LIN {X 0,Y 256.536,Z 513.805,A -85,B 0,C 180,E1 -18432.463,E2 -18432.463} C_VEL
LIN {X 0,Y 255.178,Z 520.285,A -85,B 0,C 180,E1 -18435.65,E2 -18435.65} C_VEL
LIN {X 0,Y 254.431,Z 525.317,A -85,B 0,C 180,E1 -18438.853,E2 -18438.853} C_VEL
LIN {X 0,Y 254.375,Z 529.039,A -85,B 0,C 180,E1 -18442.062,E2 -18442.062} C_VEL
LIN {X 0,Y 254.585,Z 531.508,A -85,B 0,C 180,E1 -18445.252,E2 -18445.252} C_VEL
LIN {X 0,Y 254.898,Z 532.764,A -85,B 0,C 180,E1 -18448.422,E2 -18448.422} C_VEL
LIN {X 0,Y 254.986,Z 532.93,A -85,B 0,C 180,E1 -18450.002,E2 -18450.002} C_VEL
LIN {X 0,Y 254.897,Z 532.761,A -85,B 0,C 180,E1 -18451.582,E2 -18451.582} C_VEL
LIN {X 0,Y 254.605,Z 531.496,A -85,B 0,C 180,E1 -18454.752,E2 -18454.752} C_VEL
LIN {X 0,Y 254.565,Z 530.416,A -85,B 0,C 180,E1 -18456.342,E2 -18456.342} C_VEL
LIN {X 0,Y 254.406,Z 527.304,A -85,B 0,C 180,E1 -18459.543,E2 -18459.543} C_VEL
LIN {X 0,Y 254.778,Z 522.916,A -85,B 0,C 180,E1 -18462.751,E2 -18462.751} C_VEL
LIN {X 0,Y 255.788,Z 517.161,A -85,B 0,C 180,E1 -18465.95,E2 -18465.95} C_VEL
LIN {X 0,Y 257.512,Z 509.888,A -85,B 0,C 180,E1 -18469.119,E2 -18469.119} C_VEL
LIN {X 0,Y 259.708,Z 502.128,A -85,B 0,C 180,E1 -18471.847,E2 -18471.847} C_VEL
LIN {X 0,Y 262.386,Z 492.608,A -85,B 0,C 180,E1 -18474.585,E2 -18474.585} C_VEL
LIN {X 0,Y 264.113,Z 486.805,A -85,B 0,C 180,E1 -18476.046,E2 -18476.046} C_VEL
LIN {X 0,Y 268.171,Z 478.576,A -85,B 0,C 180,E1 -18478.575,E2 -18478.575} C_VEL
LIN {X 0,Y 272.785,Z 469.047,A -85,B 0,C 180,E1 -18481.018,E2 -18481.018} C_VEL
LIN {X 0,Y 278.417,Z 457.827,A -85,B 0,C 180,E1 -18483.302,E2 -18483.302} C_VEL
LIN {X 0,Y 283.318,Z 447.662,A -85,B 0,C 180,E1 -18485.029,E2 -18485.029} C_VEL
LIN {X 0,Y 289.052,Z 435.031,A -85,B 0,C 180,E1 -18486.781,E2 -18486.781} C_VEL
LIN {X 0,Y 294.359,Z 422.603,A -85,B 0,C 180,E1 -18488.156,E2 -18488.156} C_VEL
LIN {X 0,Y 300.783,Z 405.935,A -85,B 0,C 180,E1 -18489.592,E2 -18489.592} C_VEL
LIN {X 0,Y 305.874,Z 390.525,A -85,B 0,C 180,E1 -18490.616,E2 -18490.616} C_VEL
LIN {X 0,Y 310.657,Z 373.123,A -85,B 0,C 180,E1 -18491.487,E2 -18491.487} C_VEL
LIN {X 0,Y 327.276,Z 296.354,A -85,B 0,C 180,E1 -18494.561,E2 -18494.561} C_VEL
LIN {X 0,Y 328.249,Z 291.917,A -85,B 0,C 180,E1 -18494.78,E2 -18494.78} C_VEL
LIN {X 0,Y 329.621,Z 284.935,A -85,B 0,C 180,E1 -18495.368,E2 -18495.368} C_VEL
LIN {X 0,Y 329.028,Z 283.211,A -85,B 0,C 180,E1 -18497.15,E2 -18497.15} C_VEL
LIN {X 0,Y 328.897,Z 282.812,A -85,B 0,C 180,E1 -18498.516,E2 -18498.516} C_VEL
LIN {X 0,Y 328.979,Z 283.074,A -85,B 0,C 180,E1 -18499.587,E2 -18499.587} C_VEL
LIN {X 0,Y 329.408,Z 285.035,A -85,B 0,C 180,E1 -18501.432,E2 -18501.432} C_VEL
LIN {X 0,Y 316.44,Z 338.458,A -85,B 0,C 180,E1 -18503.875,E2 -18503.875} C_VEL
LIN {X 0,Y 312.736,Z 355.057,A -85,B 0,C 180,E1 -18504.791,E2 -18504.791} C_VEL
LIN {X 0,Y 309.152,Z 368.459,A -85,B 0,C 180,E1 -18505.761,E2 -18505.761} C_VEL
LIN {X 0,Y 305.253,Z 380.868,A -85,B 0,C 180,E1 -18506.878,E2 -18506.878} C_VEL
LIN {X 0,Y 300.146,Z 394.54,A -85,B 0,C 180,E1 -18508.405,E2 -18508.405} C_VEL
LIN {X 0,Y 295.293,Z 405.891,A -85,B 0,C 180,E1 -18510.013,E2 -18510.013} C_VEL
LIN {X 0,Y 290.344,Z 416.322,A -85,B 0,C 180,E1 -18511.835,E2 -18511.835} C_VEL
LIN {X 0,Y 284.968,Z 426.311,A -85,B 0,C 180,E1 -18514.039,E2 -18514.039} C_VEL
LIN {X 0,Y 280.137,Z 434.422,A -85,B 0,C 180,E1 -18516.334,E2 -18516.334} C_VEL
LIN {X 0,Y 276.27,Z 440.16,A -85,B 0,C 180,E1 -18518.355,E2 -18518.355} C_VEL
LIN {X 0,Y 272.687,Z 444.824,A -85,B 0,C 180,E1 -18520.425,E2 -18520.425} C_VEL
LIN {X 0,Y 269.52,Z 448.489,A -85,B 0,C 180,E1 -18522.55,E2 -18522.55} C_VEL
LIN {X 0,Y 266.631,Z 451.245,A -85,B 0,C 180,E1 -18524.717,E2 -18524.717} C_VEL
LIN {X 0,Y 264.88,Z 452.58,A -85,B 0,C 180,E1 -18526.185,E2 -18526.185} C_VEL
LIN {X 0,Y 261.942,Z 454.063,A -85,B 0,C 180,E1 -18529.175,E2 -18529.175} C_VEL
LIN {X 0,Y 260.72,Z 454.217,A -85,B 0,C 180,E1 -18530.692,E2 -18530.692} C_VEL
LIN {X 0,Y 259.691,Z 453.95,A -85,B 0,C 180,E1 -18532.223,E2 -18532.223} C_VEL
LIN {X 0,Y 258.915,Z 453.273,A -85,B 0,C 180,E1 -18533.767,E2 -18533.767} C_VEL
LIN {X 0,Y 258.057,Z 452.243,A -85,B 0,C 180,E1 -18535.314,E2 -18535.314} C_VEL
LIN {X 0,Y 257.5,Z 450.798,A -85,B 0,C 180,E1 -18536.871,E2 -18536.871} C_VEL
LIN {X 0,Y 256.669,Z 447.86,A -85,B 0,C 180,E1 -18539.216,E2 -18539.216} C_VEL
LIN {X 0,Y 256.295,Z 443.931,A -85,B 0,C 180,E1 -18541.572,E2 -18541.572} C_VEL
LIN {X 0,Y 256.126,Z 438.953,A -85,B 0,C 180,E1 -18543.934,E2 -18543.934} C_VEL
LIN {X 0,Y 256.246,Z 431.674,A -85,B 0,C 180,E1 -18546.694,E2 -18546.694} C_VEL
LIN {X 0,Y 256.653,Z 423.961,A -85,B 0,C 180,E1 -18549.059,E2 -18549.059} C_VEL
LIN {X 0,Y 257.214,Z 414.588,A -85,B 0,C 180,E1 -18551.426,E2 -18551.426} C_VEL
LIN {X 0,Y 258.041,Z 403.213,A -85,B 0,C 180,E1 -18553.787,E2 -18553.787} C_VEL
LIN {X 0,Y 258.858,Z 391.632,A -85,B 0,C 180,E1 -18555.754,E2 -18555.754} C_VEL
LIN {X 0,Y 259.874,Z 379.093,A -85,B 0,C 180,E1 -18557.51,E2 -18557.51} C_VEL
LIN {X 0,Y 260.674,Z 367.212,A -85,B 0,C 180,E1 -18558.877,E2 -18558.877} C_VEL
LIN {X 0,Y 261.421,Z 353.444,A -85,B 0,C 180,E1 -18560.145,E2 -18560.145} C_VEL
LIN {X 0,Y 262.078,Z 338.203,A -85,B 0,C 180,E1 -18561.225,E2 -18561.225} C_VEL
LIN {X 0,Y 262.902,Z 318.351,A -85,B 0,C 180,E1 -18562.185,E2 -18562.185} C_VEL
LIN {X 0,Y 266.851,Z 236.98,A -85,B 0,C 180,E1 -18565.669,E2 -18565.669} C_VEL
LIN {X 0,Y 263.629,Z 209.974,A -85,B 0,C 180,E1 -18567.087,E2 -18567.087} C_VEL
LIN {X 0,Y 263.411,Z 206.92,A -85,B 0,C 180,E1 -18567.274,E2 -18567.274} C_VEL
LIN {X 0,Y 263.717,Z 203.783,A -85,B 0,C 180,E1 -18568.09,E2 -18568.09} C_VEL
LIN {X 0,Y 261.466,Z 193.257,A -85,B 0,C 180,E1 -18571.159,E2 -18571.159} C_VEL
LIN {X 0,Y 258.802,Z 181.374,A -85,B 0,C 180,E1 -18574.77,E2 -18574.77} C_VEL
LIN {X 0,Y 256.106,Z 170.203,A -85,B 0,C 180,E1 -18578.385,E2 -18578.385} C_VEL
LIN {X 0,Y 256.11,Z 170.286,A -85,B 0,C 180,E1 -18579.018,E2 -18579.018} C_VEL
LIN {X 0,Y 256.597,Z 172.135,A -85,B 0,C 180,E1 -18579.554,E2 -18579.554} C_VEL
LIN {X 0,Y 260.268,Z 178.847,A -85,B 0,C 180,E1 -18581.938,E2 -18581.938} C_VEL
LIN {X 0,Y 261.702,Z 181.55,A -85,B 0,C 180,E1 -18582.76,E2 -18582.76} C_VEL
LIN {X 0,Y 270.517,Z 194.274,A -85,B 0,C 180,E1 -18585.248,E2 -18585.248} C_VEL
LIN {X 0,Y 279.32,Z 208.41,A -85,B 0,C 180,E1 -18587.531,E2 -18587.531} C_VEL
LIN {X 0,Y 286.827,Z 222.154,A -85,B 0,C 180,E1 -18589.362,E2 -18589.362} C_VEL
LIN {X 0,Y 292.137,Z 233.078,A -85,B 0,C 180,E1 -18590.609,E2 -18590.609} C_VEL
LIN {X 0,Y 289.881,Z 285.461,A -85,B 0,C 180,E1 -18591.886,E2 -18591.886} C_VEL
LIN {X 0,Y 287.05,Z 347.338,A -85,B 0,C 180,E1 -18593.413,E2 -18593.413} C_VEL
LIN {X 0,Y 285.801,Z 362.815,A -85,B 0,C 180,E1 -18594.05,E2 -18594.05} C_VEL
LIN {X 0,Y 284.285,Z 376.98,A -85,B 0,C 180,E1 -18594.916,E2 -18594.916} C_VEL
LIN {X 0,Y 282.448,Z 389.981,A -85,B 0,C 180,E1 -18595.952,E2 -18595.952} C_VEL
LIN {X 0,Y 279.884,Z 403.781,A -85,B 0,C 180,E1 -18597.323,E2 -18597.323} C_VEL
LIN {X 0,Y 277.145,Z 416.382,A -85,B 0,C 180,E1 -18598.888,E2 -18598.888} C_VEL
LIN {X 0,Y 274.351,Z 427.21,A -85,B 0,C 180,E1 -18600.495,E2 -18600.495} C_VEL
LIN {X 0,Y 271.688,Z 436.967,A -85,B 0,C 180,E1 -18602.248,E2 -18602.248} C_VEL
LIN {X 0,Y 268.811,Z 447.132,A -85,B 0,C 180,E1 -18604.442,E2 -18604.442} C_VEL
LIN {X 0,Y 265.582,Z 457.069,A -85,B 0,C 180,E1 -18607.023,E2 -18607.023} C_VEL
LIN {X 0,Y 262.901,Z 465.292,A -85,B 0,C 180,E1 -18609.662,E2 -18609.662} C_VEL
LIN {X 0,Y 260.94,Z 471.23,A -85,B 0,C 180,E1 -18611.955,E2 -18611.955} C_VEL
LIN {X 0,Y 258.75,Z 477.709,A -85,B 0,C 180,E1 -18615.045,E2 -18615.045} C_VEL
LIN {X 0,Y 257.175,Z 482.759,A -85,B 0,C 180,E1 -18618.171,E2 -18618.171} C_VEL
LIN {X 0,Y 256.121,Z 486.236,A -85,B 0,C 180,E1 -18621.059,E2 -18621.059} C_VEL
LIN {X 0,Y 255.418,Z 488.505,A -85,B 0,C 180,E1 -18623.679,E2 -18623.679} C_VEL
LIN {X 0,Y 255.12,Z 490.193,A -85,B 0,C 180,E1 -18626.84,E2 -18626.84} C_VEL
LIN {X 0,Y 254.856,Z 490.791,A -85,B 0,C 180,E1 -18629.998,E2 -18629.998} C_VEL
LIN {X 0,Y 255.117,Z 490.228,A -85,B 0,C 180,E1 -18633.156,E2 -18633.156} C_VEL
LIN {X 0,Y 255.396,Z 488.589,A -85,B 0,C 180,E1 -18636.317,E2 -18636.317} C_VEL
LIN {X 0,Y 256.28,Z 485.793,A -85,B 0,C 180,E1 -18639.468,E2 -18639.468} C_VEL
LIN {X 0,Y 257.491,Z 481.794,A -85,B 0,C 180,E1 -18642.61,E2 -18642.61} C_VEL
LIN {X 0,Y 259.2,Z 476.467,A -85,B 0,C 180,E1 -18645.73,E2 -18645.73} C_VEL
LIN {X 0,Y 261.529,Z 469.654,A -85,B 0,C 180,E1 -18648.81,E2 -18648.81} C_VEL
LIN {X 0,Y 263.766,Z 462.707,A -85,B 0,C 180,E1 -18651.367,E2 -18651.367} C_VEL
LIN {X 0,Y 266.828,Z 453.521,A -85,B 0,C 180,E1 -18654.093,E2 -18654.093} C_VEL
LIN {X 0,Y 269.685,Z 444.479,A -85,B 0,C 180,E1 -18656.294,E2 -18656.294} C_VEL
LIN {X 0,Y 272.779,Z 433.405,A -85,B 0,C 180,E1 -18658.548,E2 -18658.548} C_VEL
LIN {X 0,Y 276.079,Z 420.918,A -85,B 0,C 180,E1 -18660.603,E2 -18660.603} C_VEL
LIN {X 0,Y 279.19,Z 407.788,A -85,B 0,C 180,E1 -18662.336,E2 -18662.336} C_VEL
LIN {X 0,Y 282.032,Z 393.095,A -85,B 0,C 180,E1 -18663.885,E2 -18663.885} C_VEL
LIN {X 0,Y 284.084,Z 379.46,A -85,B 0,C 180,E1 -18665.029,E2 -18665.029} C_VEL
LIN {X 0,Y 285.771,Z 364.638,A -85,B 0,C 180,E1 -18665.972,E2 -18665.972} C_VEL
LIN {X 0,Y 287.032,Z 349.395,A -85,B 0,C 180,E1 -18666.64,E2 -18666.64} C_VEL
LIN {X 0,Y 288.549,Z 317.716,A -85,B 0,C 180,E1 -18667.453,E2 -18667.453} C_VEL
LIN {X 0,Y 292.362,Z 233.432,A -85,B 0,C 180,E1 -18669.476,E2 -18669.476} C_VEL
LIN {X 0,Y 284.919,Z 218.308,A -85,B 0,C 180,E1 -18671.239,E2 -18671.239} C_VEL
LIN {X 0,Y 275.639,Z 202.212,A -85,B 0,C 180,E1 -18673.55,E2 -18673.55} C_VEL
LIN {X 0,Y 270.298,Z 193.85,A -85,B 0,C 180,E1 -18674.963,E2 -18674.963} C_VEL
LIN {X 0,Y 266.031,Z 189.676,A -85,B 0,C 180,E1 -18676.072,E2 -18676.072} C_VEL
LIN {X 0,Y 256.851,Z 183.256,A -85,B 0,C 180,E1 -18678.535,E2 -18678.535} C_VEL
LIN {X 0,Y 254.125,Z 180.724,A -85,B 0,C 180,E1 -18679.562,E2 -18679.562} C_VEL
LIN {X 0,Y 253.472,Z 179.796,A -85,B 0,C 180,E1 -18679.924,E2 -18679.924} C_VEL
LIN {X 0,Y 251.742,Z 176.765,A -85,B 0,C 180,E1 -18681.087,E2 -18681.087} C_VEL
LIN {X 0,Y 251.149,Z 175.254,A -85,B 0,C 180,E1 -18681.581,E2 -18681.581} C_VEL
LIN {X 0,Y 249.787,Z 173.342,A -85,B 0,C 180,E1 -18682.444,E2 -18682.444} C_VEL
LIN {X 0,Y 249.075,Z 171.086,A -85,B 0,C 180,E1 -18683.245,E2 -18683.245} C_VEL
LIN {X 0,Y 249.028,Z 171.092,A -85,B 0,C 180,E1 -18687.574,E2 -18687.574} C_VEL
LIN {X 0,Y 249.092,Z 171.068,A -85,B 0,C 180,E1 -18691.338,E2 -18691.338} C_VEL
LIN {X 0,Y 249.143,Z 171.053,A -85,B 0,C 180,E1 -18694.967,E2 -18694.967} C_VEL
LIN {X 0,Y 249.1,Z 171.058,A -85,B 0,C 180,E1 -18700.21,E2 -18700.21} C_VEL
LIN {X 0,Y 249.232,Z 171.066,A -85,B 0,C 180,E1 -18703.621,E2 -18703.621} C_VEL
LIN {X 0,Y 249.243,Z 171.046,A -85,B 0,C 180,E1 -18708.616,E2 -18708.616} C_VEL
LIN {X 0,Y 249.474,Z 171.016,A -85,B 0,C 180,E1 -18711.902,E2 -18711.902} C_VEL
LIN {X 0,Y 249.428,Z 171.042,A -85,B 0,C 180,E1 -18716.769,E2 -18716.769} C_VEL
LIN {X 0,Y 249.726,Z 170.971,A -85,B 0,C 180,E1 -18720,E2 -18720} C_VEL
LIN {X 0,Y 249.428,Z 171.039,A -85,B 0,C 180,E1 -18723.23,E2 -18723.23} C_VEL
LIN {X 0,Y 249.471,Z 171.009,A -85,B 0,C 180,E1 -18728.097,E2 -18728.097} C_VEL
LIN {X 0,Y 249.242,Z 171.043,A -85,B 0,C 180,E1 -18731.384,E2 -18731.384} C_VEL
LIN {X 0,Y 249.232,Z 171.059,A -85,B 0,C 180,E1 -18736.379,E2 -18736.379} C_VEL
LIN {X 0,Y 249.077,Z 171.081,A -85,B 0,C 180,E1 -18741.519,E2 -18741.519} C_VEL
LIN {X 0,Y 249.121,Z 171.059,A -85,B 0,C 180,E1 -18745.483,E2 -18745.483} C_VEL
LIN {X 0,Y 249.064,Z 171.067,A -85,B 0,C 180,E1 -18748.99,E2 -18748.99} C_VEL
LIN {X 0,Y 249.027,Z 171.089,A -85,B 0,C 180,E1 -18752.426,E2 -18752.426} C_VEL
LIN {X 0,Y 249.075,Z 171.201,A -85,B 0,C 180,E1 -18755.337,E2 -18755.337} C_VEL
LIN {X 0,Y 250.086,Z 173.976,A -85,B 0,C 180,E1 -18755.994,E2 -18755.994} C_VEL
LIN {X 0,Y 252.285,Z 176.508,A -85,B 0,C 180,E1 -18756.961,E2 -18756.961} C_VEL
LIN {X 0,Y 254.239,Z 179.879,A -85,B 0,C 180,E1 -18757.912,E2 -18757.912} C_VEL
LIN {X 0,Y 255.171,Z 180.942,A -85,B 0,C 180,E1 -18758.294,E2 -18758.294} C_VEL
LIN {X 0,Y 257.569,Z 184.851,A -85,B 0,C 180,E1 -18759.375,E2 -18759.375} C_VEL
LIN {X 0,Y 262.205,Z 192.372,A -85,B 0,C 180,E1 -18761.319,E2 -18761.319} C_VEL
LIN {X 0,Y 268.243,Z 209.605,A -85,B 0,C 180,E1 -18764.298,E2 -18764.298} C_VEL
LIN {X 0,Y 276.939,Z 230.172,A -85,B 0,C 180,E1 -18766.8,E2 -18766.8} C_VEL
LIN {X 0,Y 280.418,Z 238.915,A -85,B 0,C 180,E1 -18767.748,E2 -18767.748} C_VEL
LIN {X 0,Y 283.617,Z 279.318,A -85,B 0,C 180,E1 -18769.64,E2 -18769.64} C_VEL
LIN {X 0,Y 284.027,Z 287.147,A -85,B 0,C 180,E1 -18769.961,E2 -18769.961} C_VEL
LIN {X 0,Y 279.389,Z 384.707,A -85,B 0,C 180,E1 -18772.356,E2 -18772.356} C_VEL
LIN {X 0,Y 277.918,Z 399.648,A -85,B 0,C 180,E1 -18772.92,E2 -18772.92} C_VEL
LIN {X 0,Y 275.926,Z 413.694,A -85,B 0,C 180,E1 -18773.69,E2 -18773.69} C_VEL
LIN {X 0,Y 273.424,Z 427.201,A -85,B 0,C 180,E1 -18774.669,E2 -18774.669} C_VEL
LIN {X 0,Y 270.251,Z 441.425,A -85,B 0,C 180,E1 -18776.008,E2 -18776.008} C_VEL
LIN {X 0,Y 266.93,Z 454.852,A -85,B 0,C 180,E1 -18777.634,E2 -18777.634} C_VEL
LIN {X 0,Y 263.299,Z 467.497,A -85,B 0,C 180,E1 -18779.528,E2 -18779.528} C_VEL
LIN {X 0,Y 260.358,Z 477.557,A -85,B 0,C 180,E1 -18781.374,E2 -18781.374} C_VEL
LIN {X 0,Y 257.208,Z 487.833,A -85,B 0,C 180,E1 -18783.642,E2 -18783.642} C_VEL
LIN {X 0,Y 254.163,Z 497.892,A -85,B 0,C 180,E1 -18786.365,E2 -18786.365} C_VEL
LIN {X 0,Y 251.623,Z 506.261,A -85,B 0,C 180,E1 -18789.14,E2 -18789.14} C_VEL
LIN {X 0,Y 249.667,Z 513.212,A -85,B 0,C 180,E1 -18791.965,E2 -18791.965} C_VEL
LIN {X 0,Y 248.228,Z 519.693,A -85,B 0,C 180,E1 -18795.24,E2 -18795.24} C_VEL
LIN {X 0,Y 247.381,Z 524.724,A -85,B 0,C 180,E1 -18798.532,E2 -18798.532} C_VEL
LIN {X 0,Y 247.292,Z 528.448,A -85,B 0,C 180,E1 -18801.833,E2 -18801.833} C_VEL
LIN {X 0,Y 247.514,Z 530.922,A -85,B 0,C 180,E1 -18805.116,E2 -18805.116} C_VEL
LIN {X 0,Y 247.811,Z 532.178,A -85,B 0,C 180,E1 -18808.377,E2 -18808.377} C_VEL
LIN {X 0,Y 247.925,Z 532.347,A -85,B 0,C 180,E1 -18810.002,E2 -18810.002} C_VEL
LIN {X 0,Y 247.81,Z 532.175,A -85,B 0,C 180,E1 -18811.627,E2 -18811.627} C_VEL
LIN {X 0,Y 247.537,Z 530.909,A -85,B 0,C 180,E1 -18814.888,E2 -18814.888} C_VEL
LIN {X 0,Y 247.462,Z 529.824,A -85,B 0,C 180,E1 -18816.525,E2 -18816.525} C_VEL
LIN {X 0,Y 247.321,Z 526.709,A -85,B 0,C 180,E1 -18819.819,E2 -18819.819} C_VEL
LIN {X 0,Y 247.763,Z 522.321,A -85,B 0,C 180,E1 -18823.118,E2 -18823.118} C_VEL
LIN {X 0,Y 248.883,Z 516.567,A -85,B 0,C 180,E1 -18826.404,E2 -18826.404} C_VEL
LIN {X 0,Y 250.729,Z 509.294,A -85,B 0,C 180,E1 -18829.657,E2 -18829.657} C_VEL
LIN {X 0,Y 253.013,Z 501.532,A -85,B 0,C 180,E1 -18832.456,E2 -18832.456} C_VEL
LIN {X 0,Y 255.792,Z 492.22,A -85,B 0,C 180,E1 -18835.207,E2 -18835.207} C_VEL
LIN {X 0,Y 256.925,Z 488.661,A -85,B 0,C 180,E1 -18836.175,E2 -18836.175} C_VEL
LIN {X 0,Y 261.341,Z 480.431,A -85,B 0,C 180,E1 -18838.953,E2 -18838.953} C_VEL
LIN {X 0,Y 266.061,Z 471.495,A -85,B 0,C 180,E1 -18841.448,E2 -18841.448} C_VEL
LIN {X 0,Y 271.832,Z 461.11,A -85,B 0,C 180,E1 -18843.772,E2 -18843.772} C_VEL
LIN {X 0,Y 277.172,Z 450.863,A -85,B 0,C 180,E1 -18845.677,E2 -18845.677} C_VEL
LIN {X 0,Y 283.089,Z 439.038,A -85,B 0,C 180,E1 -18847.464,E2 -18847.464} C_VEL
LIN {X 0,Y 289.615,Z 425.159,A -85,B 0,C 180,E1 -18849.121,E2 -18849.121} C_VEL
LIN {X 0,Y 296.704,Z 408.403,A -85,B 0,C 180,E1 -18850.648,E2 -18850.648} C_VEL
LIN {X 0,Y 302.336,Z 393.002,A -85,B 0,C 180,E1 -18851.715,E2 -18851.715} C_VEL
LIN {X 0,Y 307.881,Z 374.881,A -85,B 0,C 180,E1 -18852.664,E2 -18852.664} C_VEL
LIN {X 0,Y 313.284,Z 351.402,A -85,B 0,C 180,E1 -18853.632,E2 -18853.632} C_VEL
LIN {X 0,Y 326.613,Z 294.43,A -85,B 0,C 180,E1 -18855.907,E2 -18855.907} C_VEL
LIN {X 0,Y 327.357,Z 290.873,A -85,B 0,C 180,E1 -18856.23,E2 -18856.23} C_VEL
LIN {X 0,Y 327.092,Z 289.871,A -85,B 0,C 180,E1 -18857.46,E2 -18857.46} C_VEL
LIN {X 0,Y 327.032,Z 289.726,A -85,B 0,C 180,E1 -18859.296,E2 -18859.296} C_VEL
LIN {X 0,Y 327.104,Z 290.812,A -85,B 0,C 180,E1 -18860.396,E2 -18860.396} C_VEL
LIN {X 0,Y 313.508,Z 344.767,A -85,B 0,C 180,E1 -18862.903,E2 -18862.903} C_VEL
LIN {X 0,Y 310.152,Z 358.542,A -85,B 0,C 180,E1 -18863.702,E2 -18863.702} C_VEL
LIN {X 0,Y 305.497,Z 374.231,A -85,B 0,C 180,E1 -18864.892,E2 -18864.892} C_VEL
LIN {X 0,Y 300.968,Z 386.739,A -85,B 0,C 180,E1 -18866.116,E2 -18866.116} C_VEL
LIN {X 0,Y 295.592,Z 399.622,A -85,B 0,C 180,E1 -18867.659,E2 -18867.659} C_VEL
LIN {X 0,Y 290.065,Z 411.145,A -85,B 0,C 180,E1 -18869.416,E2 -18869.416} C_VEL
LIN {X 0,Y 284.888,Z 420.753,A -85,B 0,C 180,E1 -18871.246,E2 -18871.246} C_VEL
LIN {X 0,Y 280.059,Z 428.908,A -85,B 0,C 180,E1 -18873.147,E2 -18873.147} C_VEL
LIN {X 0,Y 275.65,Z 435.696,A -85,B 0,C 180,E1 -18875.122,E2 -18875.122} C_VEL
LIN {X 0,Y 271.474,Z 441.357,A -85,B 0,C 180,E1 -18877.15,E2 -18877.15} C_VEL
LIN {X 0,Y 267.638,Z 446.047,A -85,B 0,C 180,E1 -18879.237,E2 -18879.237} C_VEL
LIN {X 0,Y 264.173,Z 449.709,A -85,B 0,C 180,E1 -18881.383,E2 -18881.383} C_VEL
LIN {X 0,Y 260.072,Z 453.216,A -85,B 0,C 180,E1 -18884.322,E2 -18884.322} C_VEL
LIN {X 0,Y 258.236,Z 454.39,A -85,B 0,C 180,E1 -18885.822,E2 -18885.822} C_VEL
LIN {X 0,Y 255.125,Z 455.511,A -85,B 0,C 180,E1 -18888.882,E2 -18888.882} C_VEL
LIN {X 0,Y 253.832,Z 455.496,A -85,B 0,C 180,E1 -18890.438,E2 -18890.438} C_VEL
LIN {X 0,Y 251.953,Z 454.272,A -85,B 0,C 180,E1 -18893.594,E2 -18893.594} C_VEL
LIN {X 0,Y 251.059,Z 453.11,A -85,B 0,C 180,E1 -18895.183,E2 -18895.183} C_VEL
LIN {X 0,Y 250.13,Z 450.551,A -85,B 0,C 180,E1 -18897.585,E2 -18897.585} C_VEL
LIN {X 0,Y 249.344,Z 447.068,A -85,B 0,C 180,E1 -18900,E2 -18900} C_VEL
LIN {X 0,Y 249.111,Z 442.563,A -85,B 0,C 180,E1 -18902.426,E2 -18902.426} C_VEL
LIN {X 0,Y 249.031,Z 435.932,A -85,B 0,C 180,E1 -18905.263,E2 -18905.263} C_VEL
LIN {X 0,Y 249.417,Z 427.545,A -85,B 0,C 180,E1 -18908.099,E2 -18908.099} C_VEL
LIN {X 0,Y 249.843,Z 418.719,A -85,B 0,C 180,E1 -18910.535,E2 -18910.535} C_VEL
LIN {X 0,Y 250.622,Z 408.042,A -85,B 0,C 180,E1 -18912.964,E2 -18912.964} C_VEL
LIN {X 0,Y 251.508,Z 396.079,A -85,B 0,C 180,E1 -18915.187,E2 -18915.187} C_VEL
LIN {X 0,Y 252.395,Z 384.282,A -85,B 0,C 180,E1 -18917,E2 -18917} C_VEL
LIN {X 0,Y 253.536,Z 369.719,A -85,B 0,C 180,E1 -18918.799,E2 -18918.799} C_VEL
LIN {X 0,Y 254.275,Z 355.561,A -85,B 0,C 180,E1 -18920.189,E2 -18920.189} C_VEL
LIN {X 0,Y 255.037,Z 339.802,A -85,B 0,C 180,E1 -18921.363,E2 -18921.363} C_VEL
LIN {X 0,Y 255.684,Z 323.748,A -85,B 0,C 180,E1 -18922.207,E2 -18922.207} C_VEL
LIN {X 0,Y 259.997,Z 238.073,A -85,B 0,C 180,E1 -18926.006,E2 -18926.006} C_VEL
LIN {X 0,Y 256.816,Z 210.902,A -85,B 0,C 180,E1 -18927.469,E2 -18927.469} C_VEL
LIN {X 0,Y 256.568,Z 207.28,A -85,B 0,C 180,E1 -18927.683,E2 -18927.683} C_VEL
LIN {X 0,Y 256.729,Z 204.889,A -85,B 0,C 180,E1 -18928.328,E2 -18928.328} C_VEL
LIN {X 0,Y 254.286,Z 193.66,A -85,B 0,C 180,E1 -18931.677,E2 -18931.677} C_VEL
LIN {X 0,Y 252.016,Z 183.382,A -85,B 0,C 180,E1 -18934.868,E2 -18934.868} C_VEL
LIN {X 0,Y 249.804,Z 174.098,A -85,B 0,C 180,E1 -18937.921,E2 -18937.921} C_VEL
LIN {X 0,Y 251.531,Z 176.347,A -85,B 0,C 180,E1 -18938.952,E2 -18938.952} C_VEL
LIN {X 0,Y 254.556,Z 182.21,A -85,B 0,C 180,E1 -18940.987,E2 -18940.987} C_VEL
LIN {X 0,Y 260.072,Z 189.785,A -85,B 0,C 180,E1 -18942.697,E2 -18942.697} C_VEL
LIN {X 0,Y 267.015,Z 199.952,A -85,B 0,C 180,E1 -18944.701,E2 -18944.701} C_VEL
LIN {X 0,Y 275.207,Z 213.371,A -85,B 0,C 180,E1 -18946.904,E2 -18946.904} C_VEL
LIN {X 0,Y 282.388,Z 226.708,A -85,B 0,C 180,E1 -18948.723,E2 -18948.723} C_VEL
LIN {X 0,Y 286.681,Z 235.63,A -85,B 0,C 180,E1 -18949.775,E2 -18949.775} C_VEL
LIN {X 0,Y 283.811,Z 296.33,A -85,B 0,C 180,E1 -18951.25,E2 -18951.25} C_VEL
LIN {X 0,Y 281.398,Z 347.863,A -85,B 0,C 180,E1 -18952.554,E2 -18952.554} C_VEL
LIN {X 0,Y 280.165,Z 362.884,A -85,B 0,C 180,E1 -18953.178,E2 -18953.178} C_VEL
LIN {X 0,Y 278.675,Z 376.502,A -85,B 0,C 180,E1 -18954.009,E2 -18954.009} C_VEL
LIN {X 0,Y 276.62,Z 390.551,A -85,B 0,C 180,E1 -18955.133,E2 -18955.133} C_VEL
LIN {X 0,Y 273.976,Z 404.354,A -85,B 0,C 180,E1 -18956.527,E2 -18956.527} C_VEL
LIN {X 0,Y 271.126,Z 416.958,A -85,B 0,C 180,E1 -18958.118,E2 -18958.118} C_VEL
LIN {X 0,Y 268.208,Z 427.791,A -85,B 0,C 180,E1 -18959.749,E2 -18959.749} C_VEL
LIN {X 0,Y 265.435,Z 437.55,A -85,B 0,C 180,E1 -18961.535,E2 -18961.535} C_VEL
LIN {X 0,Y 262.446,Z 447.714,A -85,B 0,C 180,E1 -18963.776,E2 -18963.776} C_VEL
LIN {X 0,Y 259.085,Z 457.652,A -85,B 0,C 180,E1 -18966.413,E2 -18966.413} C_VEL
LIN {X 0,Y 256.26,Z 465.877,A -85,B 0,C 180,E1 -18969.111,E2 -18969.111} C_VEL
LIN {X 0,Y 254.2,Z 471.816,A -85,B 0,C 180,E1 -18971.459,E2 -18971.459} C_VEL
LIN {X 0,Y 251.917,Z 478.294,A -85,B 0,C 180,E1 -18974.629,E2 -18974.629} C_VEL
LIN {X 0,Y 250.244,Z 483.345,A -85,B 0,C 180,E1 -18977.838,E2 -18977.838} C_VEL
LIN {X 0,Y 249.111,Z 486.928,A -85,B 0,C 180,E1 -18980.908,E2 -18980.908} C_VEL
LIN {X 0,Y 248.384,Z 489.09,A -85,B 0,C 180,E1 -18983.499,E2 -18983.499} C_VEL
LIN {X 0,Y 248.079,Z 490.776,A -85,B 0,C 180,E1 -18986.75,E2 -18986.75} C_VEL
LIN {X 0,Y 247.803,Z 491.374,A -85,B 0,C 180,E1 -18989.998,E2 -18989.998} C_VEL
LIN {X 0,Y 248.076,Z 490.811,A -85,B 0,C 180,E1 -18993.246,E2 -18993.246} C_VEL
LIN {X 0,Y 248.364,Z 489.173,A -85,B 0,C 180,E1 -18996.497,E2 -18996.497} C_VEL
LIN {X 0,Y 249.293,Z 486.378,A -85,B 0,C 180,E1 -18999.736,E2 -18999.736} C_VEL
LIN {X 0,Y 250.579,Z 482.378,A -85,B 0,C 180,E1 -19002.964,E2 -19002.964} C_VEL
LIN {X 0,Y 252.388,Z 477.05,A -85,B 0,C 180,E1 -19006.166,E2 -19006.166} C_VEL
LIN {X 0,Y 254.83,Z 470.236,A -85,B 0,C 180,E1 -19009.324,E2 -19009.324} C_VEL
LIN {X 0,Y 257.302,Z 462.912,A -85,B 0,C 180,E1 -19012.065,E2 -19012.065} C_VEL
LIN {X 0,Y 260.367,Z 454.101,A -85,B 0,C 180,E1 -19014.73,E2 -19014.73} C_VEL
LIN {X 0,Y 263.36,Z 445.056,A -85,B 0,C 180,E1 -19016.976,E2 -19016.976} C_VEL
LIN {X 0,Y 266.516,Z 434.189,A -85,B 0,C 180,E1 -19019.235,E2 -19019.235} C_VEL
LIN {X 0,Y 269.713,Z 422.629,A -85,B 0,C 180,E1 -19021.188,E2 -19021.188} C_VEL
LIN {X 0,Y 272.887,Z 409.752,A -85,B 0,C 180,E1 -19022.958,E2 -19022.958} C_VEL
LIN {X 0,Y 275.522,Z 397.187,A -85,B 0,C 180,E1 -19024.355,E2 -19024.355} C_VEL
LIN {X 0,Y 277.864,Z 383.592,A -85,B 0,C 180,E1 -19025.57,E2 -19025.57} C_VEL
LIN {X 0,Y 279.622,Z 369.146,A -85,B 0,C 180,E1 -19026.593,E2 -19026.593} C_VEL
LIN {X 0,Y 281.057,Z 354.334,A -85,B 0,C 180,E1 -19027.326,E2 -19027.326} C_VEL
LIN {X 0,Y 282.01,Z 337.753,A -85,B 0,C 180,E1 -19027.853,E2 -19027.853} C_VEL
LIN {X 0,Y 286.823,Z 235.74,A -85,B 0,C 180,E1 -19030.333,E2 -19030.333} C_VEL
LIN {X 0,Y 279.234,Z 220.529,A -85,B 0,C 180,E1 -19032.21,E2 -19032.21} C_VEL
LIN {X 0,Y 270.912,Z 206.138,A -85,B 0,C 180,E1 -19034.379,E2 -19034.379} C_VEL
LIN {X 0,Y 263.553,Z 194.732,A -85,B 0,C 180,E1 -19036.436,E2 -19036.436} C_VEL
LIN {X 0,Y 256.118,Z 184.27,A -85,B 0,C 180,E1 -19038.681,E2 -19038.681} C_VEL
LIN {X 0,Y 254.314,Z 181.772,A -85,B 0,C 180,E1 -19039.284,E2 -19039.284} C_VEL
LIN {X 0,Y 253.472,Z 179.796,A -85,B 0,C 180,E1 -19039.924,E2 -19039.924} C_VEL
LIN {X 0,Y 251.945,Z 178.354,A -85,B 0,C 180,E1 -19040.686,E2 -19040.686} C_VEL
LIN {X 0,Y 248.463,Z 177.34,A -85,B 0,C 180,E1 -19041.976,E2 -19041.976} C_VEL
LIN {X 0,Y 244.957,Z 176.469,A -85,B 0,C 180,E1 -19043.305,E2 -19043.305} C_VEL
LIN {X 0,Y 243.397,Z 175.229,A -85,B 0,C 180,E1 -19044.123,E2 -19044.123} C_VEL
LIN {X 0,Y 242.265,Z 173.058,A -85,B 0,C 180,E1 -19045.044,E2 -19045.044} C_VEL
LIN {X 0,Y 242.03,Z 171.944,A -85,B 0,C 180,E1 -19045.448,E2 -19045.448} C_VEL
LIN {X 0,Y 242.03,Z 171.942,A -85,B 0,C 180,E1 -19050.585,E2 -19050.585} C_VEL
LIN {X 0,Y 242.059,Z 171.94,A -85,B 0,C 180,E1 -19054.182,E2 -19054.182} C_VEL
LIN {X 0,Y 242.044,Z 171.961,A -85,B 0,C 180,E1 -19058.296,E2 -19058.296} C_VEL
LIN {X 0,Y 242.154,Z 171.942,A -85,B 0,C 180,E1 -19063.277,E2 -19063.277} C_VEL
LIN {X 0,Y 242.176,Z 171.921,A -85,B 0,C 180,E1 -19068.279,E2 -19068.279} C_VEL
LIN {X 0,Y 242.425,Z 171.897,A -85,B 0,C 180,E1 -19071.665,E2 -19071.665} C_VEL
LIN {X 0,Y 242.251,Z 171.913,A -85,B 0,C 180,E1 -19075.007,E2 -19075.007} C_VEL
LIN {X 0,Y 242.627,Z 171.871,A -85,B 0,C 180,E1 -19078.34,E2 -19078.34} C_VEL
LIN {X 0,Y 242.627,Z 171.864,A -85,B 0,C 180,E1 -19081.66,E2 -19081.66} C_VEL
LIN {X 0,Y 242.424,Z 171.879,A -85,B 0,C 180,E1 -19086.659,E2 -19086.659} C_VEL
LIN {X 0,Y 242.304,Z 171.923,A -85,B 0,C 180,E1 -19090.022,E2 -19090.022} C_VEL
LIN {X 0,Y 242.156,Z 171.931,A -85,B 0,C 180,E1 -19095.141,E2 -19095.141} C_VEL
LIN {X 0,Y 242.063,Z 171.928,A -85,B 0,C 180,E1 -19098.625,E2 -19098.625} C_VEL
LIN {X 0,Y 242.003,Z 171.962,A -85,B 0,C 180,E1 -19102.181,E2 -19102.181} C_VEL
LIN {X 0,Y 242.057,Z 171.942,A -85,B 0,C 180,E1 -19105.839,E2 -19105.839} C_VEL
LIN {X 0,Y 241.998,Z 171.945,A -85,B 0,C 180,E1 -19109.584,E2 -19109.584} C_VEL
LIN {X 0,Y 241.973,Z 172.039,A -85,B 0,C 180,E1 -19113.015,E2 -19113.015} C_VEL
LIN {X 0,Y 243.096,Z 174.98,A -85,B 0,C 180,E1 -19113.816,E2 -19113.816} C_VEL
LIN {X 0,Y 245.408,Z 177.662,A -85,B 0,C 180,E1 -19114.943,E2 -19114.943} C_VEL
LIN {X 0,Y 247.382,Z 180.974,A -85,B 0,C 180,E1 -19115.992,E2 -19115.992} C_VEL
LIN {X 0,Y 248.404,Z 182.138,A -85,B 0,C 180,E1 -19116.452,E2 -19116.452} C_VEL
LIN {X 0,Y 250.802,Z 185.973,A -85,B 0,C 180,E1 -19117.615,E2 -19117.615} C_VEL
LIN {X 0,Y 256.362,Z 194.76,A -85,B 0,C 180,E1 -19120.107,E2 -19120.107} C_VEL
LIN {X 0,Y 257.933,Z 197.915,A -85,B 0,C 180,E1 -19120.839,E2 -19120.839} C_VEL
LIN {X 0,Y 261.667,Z 208.915,A -85,B 0,C 180,E1 -19122.799,E2 -19122.799} C_VEL
LIN {X 0,Y 267.711,Z 222.786,A -85,B 0,C 180,E1 -19124.673,E2 -19124.673} C_VEL
LIN {X 0,Y 275.279,Z 241.482,A -85,B 0,C 180,E1 -19126.874,E2 -19126.874} C_VEL
LIN {X 0,Y 278.586,Z 285.723,A -85,B 0,C 180,E1 -19128.982,E2 -19128.982} C_VEL
LIN {X 0,Y 273.991,Z 381.324,A -85,B 0,C 180,E1 -19131.363,E2 -19131.363} C_VEL
LIN {X 0,Y 272.643,Z 396.433,A -85,B 0,C 180,E1 -19131.902,E2 -19131.902} C_VEL
LIN {X 0,Y 270.644,Z 410.578,A -85,B 0,C 180,E1 -19132.63,E2 -19132.63} C_VEL
LIN {X 0,Y 268.087,Z 424.672,A -85,B 0,C 180,E1 -19133.624,E2 -19133.624} C_VEL
LIN {X 0,Y 264.757,Z 439.279,A -85,B 0,C 180,E1 -19134.97,E2 -19134.97} C_VEL
LIN {X 0,Y 261.551,Z 451.91,A -85,B 0,C 180,E1 -19136.463,E2 -19136.463} C_VEL
LIN {X 0,Y 257.911,Z 464.78,A -85,B 0,C 180,E1 -19138.364,E2 -19138.364} C_VEL
LIN {X 0,Y 254.611,Z 475.065,A -85,B 0,C 180,E1 -19140.211,E2 -19140.211} C_VEL
LIN {X 0,Y 251.289,Z 485.608,A -85,B 0,C 180,E1 -19142.521,E2 -19142.521} C_VEL
LIN {X 0,Y 248.047,Z 495.609,A -85,B 0,C 180,E1 -19145.193,E2 -19145.193} C_VEL
LIN {X 0,Y 245.288,Z 504.537,A -85,B 0,C 180,E1 -19148.134,E2 -19148.134} C_VEL
LIN {X 0,Y 242.815,Z 512.619,A -85,B 0,C 180,E1 -19151.437,E2 -19151.437} C_VEL
LIN {X 0,Y 241.265,Z 519.1,A -85,B 0,C 180,E1 -19154.804,E2 -19154.804} C_VEL
LIN {X 0,Y 240.339,Z 524.131,A -85,B 0,C 180,E1 -19158.191,E2 -19158.191} C_VEL
LIN {X 0,Y 240.189,Z 527.856,A -85,B 0,C 180,E1 -19161.59,E2 -19161.59} C_VEL
LIN {X 0,Y 240.422,Z 530.334,A -85,B 0,C 180,E1 -19164.971,E2 -19164.971} C_VEL
LIN {X 0,Y 240.726,Z 531.592,A -85,B 0,C 180,E1 -19168.329,E2 -19168.329} C_VEL
LIN {X 0,Y 240.864,Z 531.763,A -85,B 0,C 180,E1 -19170.002,E2 -19170.002} C_VEL
LIN {X 0,Y 240.726,Z 531.589,A -85,B 0,C 180,E1 -19171.675,E2 -19171.675} C_VEL
LIN {X 0,Y 240.446,Z 530.321,A -85,B 0,C 180,E1 -19175.033,E2 -19175.033} C_VEL
LIN {X 0,Y 240.352,Z 529.233,A -85,B 0,C 180,E1 -19176.719,E2 -19176.719} C_VEL
LIN {X 0,Y 240.255,Z 526.116,A -85,B 0,C 180,E1 -19180.111,E2 -19180.111} C_VEL
LIN {X 0,Y 240.761,Z 521.727,A -85,B 0,C 180,E1 -19183.507,E2 -19183.507} C_VEL
LIN {X 0,Y 241.966,Z 515.971,A -85,B 0,C 180,E1 -19186.887,E2 -19186.887} C_VEL
LIN {X 0,Y 243.937,Z 508.697,A -85,B 0,C 180,E1 -19190.228,E2 -19190.228} C_VEL
LIN {X 0,Y 246.359,Z 500.937,A -85,B 0,C 180,E1 -19193.097,E2 -19193.097} C_VEL
LIN {X 0,Y 249.546,Z 490.893,A -85,B 0,C 180,E1 -19196.109,E2 -19196.109} C_VEL
LIN {X 0,Y 254.49,Z 482.168,A -85,B 0,C 180,E1 -19199.355,E2 -19199.355} C_VEL
LIN {X 0,Y 260.101,Z 472.572,A -85,B 0,C 180,E1 -19202.254,E2 -19202.254} C_VEL
LIN {X 0,Y 266.952,Z 461.181,A -85,B 0,C 180,E1 -19204.934,E2 -19204.934} C_VEL
LIN {X 0,Y 272.592,Z 451.213,A -85,B 0,C 180,E1 -19206.831,E2 -19206.831} C_VEL
LIN {X 0,Y 278.792,Z 439.861,A -85,B 0,C 180,E1 -19208.605,E2 -19208.605} C_VEL
LIN {X 0,Y 285.563,Z 426.579,A -85,B 0,C 180,E1 -19210.246,E2 -19210.246} C_VEL
LIN {X 0,Y 292.284,Z 412.067,A -85,B 0,C 180,E1 -19211.626,E2 -19211.626} C_VEL
LIN {X 0,Y 298.69,Z 396.357,A -85,B 0,C 180,E1 -19212.787,E2 -19212.787} C_VEL
LIN {X 0,Y 303.757,Z 381.793,A -85,B 0,C 180,E1 -19213.614,E2 -19213.614} C_VEL
LIN {X 0,Y 308.669,Z 364.598,A -85,B 0,C 180,E1 -19214.383,E2 -19214.383} C_VEL
LIN {X 0,Y 325.261,Z 297.037,A -85,B 0,C 180,E1 -19217.054,E2 -19217.054} C_VEL
LIN {X 0,Y 325.113,Z 296.581,A -85,B 0,C 180,E1 -19217.923,E2 -19217.923} C_VEL
LIN {X 0,Y 325.11,Z 296.665,A -85,B 0,C 180,E1 -19219.372,E2 -19219.372} C_VEL
LIN {X 0,Y 311.551,Z 348.188,A -85,B 0,C 180,E1 -19221.762,E2 -19221.762} C_VEL
LIN {X 0,Y 307.916,Z 361.828,A -85,B 0,C 180,E1 -19222.577,E2 -19222.577} C_VEL
LIN {X 0,Y 303.582,Z 375.43,A -85,B 0,C 180,E1 -19223.614,E2 -19223.614} C_VEL
LIN {X 0,Y 298.765,Z 387.827,A -85,B 0,C 180,E1 -19224.808,E2 -19224.808} C_VEL
LIN {X 0,Y 293.069,Z 400.582,A -85,B 0,C 180,E1 -19226.32,E2 -19226.32} C_VEL
LIN {X 0,Y 286.727,Z 412.918,A -85,B 0,C 180,E1 -19228.198,E2 -19228.198} C_VEL
LIN {X 0,Y 280.367,Z 423.832,A -85,B 0,C 180,E1 -19230.325,E2 -19230.325} C_VEL
LIN {X 0,Y 274.461,Z 432.735,A -85,B 0,C 180,E1 -19232.554,E2 -19232.554} C_VEL
LIN {X 0,Y 269.834,Z 439.049,A -85,B 0,C 180,E1 -19234.548,E2 -19234.548} C_VEL
LIN {X 0,Y 265.458,Z 444.379,A -85,B 0,C 180,E1 -19236.602,E2 -19236.602} C_VEL
LIN {X 0,Y 260.162,Z 449.91,A -85,B 0,C 180,E1 -19239.441,E2 -19239.441} C_VEL
LIN {X 0,Y 255.577,Z 453.8,A -85,B 0,C 180,E1 -19242.393,E2 -19242.393} C_VEL
LIN {X 0,Y 251.576,Z 456.113,A -85,B 0,C 180,E1 -19245.438,E2 -19245.438} C_VEL
LIN {X 0,Y 248.304,Z 456.923,A -85,B 0,C 180,E1 -19248.573,E2 -19248.573} C_VEL
LIN {X 0,Y 245.836,Z 456.2,A -85,B 0,C 180,E1 -19251.782,E2 -19251.782} C_VEL
LIN {X 0,Y 244.972,Z 455.218,A -85,B 0,C 180,E1 -19253.411,E2 -19253.411} C_VEL
LIN {X 0,Y 244.042,Z 453.871,A -85,B 0,C 180,E1 -19255.044,E2 -19255.044} C_VEL
LIN {X 0,Y 243.063,Z 451.116,A -85,B 0,C 180,E1 -19257.514,E2 -19257.514} C_VEL
LIN {X 0,Y 242.253,Z 447.413,A -85,B 0,C 180,E1 -19260,E2 -19260} C_VEL
LIN {X 0,Y 242.018,Z 442.667,A -85,B 0,C 180,E1 -19262.497,E2 -19262.497} C_VEL
LIN {X 0,Y 241.949,Z 435.701,A -85,B 0,C 180,E1 -19265.417,E2 -19265.417} C_VEL
LIN {X 0,Y 242.368,Z 426.997,A -85,B 0,C 180,E1 -19268.337,E2 -19268.337} C_VEL
LIN {X 0,Y 242.834,Z 417.837,A -85,B 0,C 180,E1 -19270.843,E2 -19270.843} C_VEL
LIN {X 0,Y 243.632,Z 406.701,A -85,B 0,C 180,E1 -19273.343,E2 -19273.343} C_VEL
LIN {X 0,Y 244.486,Z 395.526,A -85,B 0,C 180,E1 -19275.421,E2 -19275.421} C_VEL
LIN {X 0,Y 245.439,Z 383.378,A -85,B 0,C 180,E1 -19277.283,E2 -19277.283} C_VEL
LIN {X 0,Y 246.46,Z 370.286,A -85,B 0,C 180,E1 -19278.927,E2 -19278.927} C_VEL
LIN {X 0,Y 247.158,Z 357.689,A -85,B 0,C 180,E1 -19280.217,E2 -19280.217} C_VEL
LIN {X 0,Y 247.934,Z 342.665,A -85,B 0,C 180,E1 -19281.405,E2 -19281.405} C_VEL
LIN {X 0,Y 248.512,Z 328.59,A -85,B 0,C 180,E1 -19282.226,E2 -19282.226} C_VEL
LIN {X 0,Y 252.287,Z 253.794,A -85,B 0,C 180,E1 -19285.692,E2 -19285.692} C_VEL
LIN {X 0,Y 252.993,Z 238.12,A -85,B 0,C 180,E1 -19286.41,E2 -19286.41} C_VEL
LIN {X 0,Y 249.846,Z 210.034,A -85,B 0,C 180,E1 -19287.96,E2 -19287.96} C_VEL
LIN {X 0,Y 249.72,Z 207.558,A -85,B 0,C 180,E1 -19288.125,E2 -19288.125} C_VEL
LIN {X 0,Y 249.263,Z 203.571,A -85,B 0,C 180,E1 -19289.278,E2 -19289.278} C_VEL
LIN {X 0,Y 245.911,Z 188.315,A -85,B 0,C 180,E1 -19294.021,E2 -19294.021} C_VEL
LIN {X 0,Y 243.75,Z 179.128,A -85,B 0,C 180,E1 -19297.084,E2 -19297.084} C_VEL
LIN {X 0,Y 246.144,Z 180.635,A -85,B 0,C 180,E1 -19298.199,E2 -19298.199} C_VEL
LIN {X 0,Y 247.847,Z 183.265,A -85,B 0,C 180,E1 -19299.184,E2 -19299.184} C_VEL
LIN {X 0,Y 256.093,Z 194.506,A -85,B 0,C 180,E1 -19301.903,E2 -19301.903} C_VEL
LIN {X 0,Y 263.154,Z 205.078,A -85,B 0,C 180,E1 -19304.029,E2 -19304.029} C_VEL
LIN {X 0,Y 271.135,Z 218.269,A -85,B 0,C 180,E1 -19306.257,E2 -19306.257} C_VEL
LIN {X 0,Y 278.075,Z 231.448,A -85,B 0,C 180,E1 -19308.087,E2 -19308.087} C_VEL
LIN {X 0,Y 281.249,Z 238.047,A -85,B 0,C 180,E1 -19308.897,E2 -19308.897} C_VEL
LIN {X 0,Y 275.829,Z 348.387,A -85,B 0,C 180,E1 -19311.662,E2 -19311.662} C_VEL
LIN {X 0,Y 274.528,Z 363.555,A -85,B 0,C 180,E1 -19312.3,E2 -19312.3} C_VEL
LIN {X 0,Y 272.903,Z 377.617,A -85,B 0,C 180,E1 -19313.175,E2 -19313.175} C_VEL
LIN {X 0,Y 270.854,Z 391.12,A -85,B 0,C 180,E1 -19314.278,E2 -19314.278} C_VEL
LIN {X 0,Y 268.12,Z 404.927,A -85,B 0,C 180,E1 -19315.696,E2 -19315.696} C_VEL
LIN {X 0,Y 265.149,Z 417.536,A -85,B 0,C 180,E1 -19317.311,E2 -19317.311} C_VEL
LIN {X 0,Y 262.126,Z 428.37,A -85,B 0,C 180,E1 -19318.971,E2 -19318.971} C_VEL
LIN {X 0,Y 258.733,Z 439.975,A -85,B 0,C 180,E1 -19321.172,E2 -19321.172} C_VEL
LIN {X 0,Y 255.553,Z 449.88,A -85,B 0,C 180,E1 -19323.454,E2 -19323.454} C_VEL
LIN {X 0,Y 252.141,Z 459.547,A -85,B 0,C 180,E1 -19326.159,E2 -19326.159} C_VEL
LIN {X 0,Y 249.267,Z 467.544,A -85,B 0,C 180,E1 -19328.93,E2 -19328.93} C_VEL
LIN {X 0,Y 246.76,Z 474.156,A -85,B 0,C 180,E1 -19331.74,E2 -19331.74} C_VEL
LIN {X 0,Y 244.591,Z 480.251,A -85,B 0,C 180,E1 -19335.011,E2 -19335.011} C_VEL
LIN {X 0,Y 242.958,Z 484.955,A -85,B 0,C 180,E1 -19338.315,E2 -19338.315} C_VEL
LIN {X 0,Y 241.819,Z 488.396,A -85,B 0,C 180,E1 -19341.642,E2 -19341.642} C_VEL
LIN {X 0,Y 241.185,Z 490.654,A -85,B 0,C 180,E1 -19344.983,E2 -19344.983} C_VEL
LIN {X 0,Y 240.823,Z 491.804,A -85,B 0,C 180,E1 -19348.326,E2 -19348.326} C_VEL
LIN {X 0,Y 240.822,Z 491.815,A -85,B 0,C 180,E1 -19351.67,E2 -19351.67} C_VEL
LIN {X 0,Y 241.171,Z 490.712,A -85,B 0,C 180,E1 -19355.013,E2 -19355.013} C_VEL
LIN {X 0,Y 241.819,Z 488.501,A -85,B 0,C 180,E1 -19358.353,E2 -19358.353} C_VEL
LIN {X 0,Y 242.937,Z 485.119,A -85,B 0,C 180,E1 -19361.681,E2 -19361.681} C_VEL
LIN {X 0,Y 244.54,Z 480.474,A -85,B 0,C 180,E1 -19364.988,E2 -19364.988} C_VEL
LIN {X 0,Y 246.707,Z 474.43,A -85,B 0,C 180,E1 -19368.259,E2 -19368.259} C_VEL
LIN {X 0,Y 249.178,Z 467.881,A -85,B 0,C 180,E1 -19371.074,E2 -19371.074} C_VEL
LIN {X 0,Y 252.08,Z 459.933,A -85,B 0,C 180,E1 -19373.842,E2 -19373.842} C_VEL
LIN {X 0,Y 255.45,Z 450.353,A -85,B 0,C 180,E1 -19376.554,E2 -19376.554} C_VEL
LIN {X 0,Y 258.593,Z 440.521,A -85,B 0,C 180,E1 -19378.84,E2 -19378.84} C_VEL
LIN {X 0,Y 261.801,Z 429.85,A -85,B 0,C 180,E1 -19380.888,E2 -19380.888} C_VEL
LIN {X 0,Y 265.004,Z 418.322,A -85,B 0,C 180,E1 -19382.705,E2 -19382.705} C_VEL
LIN {X 0,Y 268.044,Z 405.864,A -85,B 0,C 180,E1 -19384.311,E2 -19384.311} C_VEL
LIN {X 0,Y 270.748,Z 392.294,A -85,B 0,C 180,E1 -19385.733,E2 -19385.733} C_VEL
LIN {X 0,Y 272.976,Z 377.845,A -85,B 0,C 180,E1 -19386.93,E2 -19386.93} C_VEL
LIN {X 0,Y 274.729,Z 363.263,A -85,B 0,C 180,E1 -19387.824,E2 -19387.824} C_VEL
LIN {X 0,Y 275.964,Z 347.612,A -85,B 0,C 180,E1 -19388.485,E2 -19388.485} C_VEL
LIN {X 0,Y 281.372,Z 239.336,A -85,B 0,C 180,E1 -19391.177,E2 -19391.177} C_VEL
LIN {X 0,Y 281.108,Z 237.621,A -85,B 0,C 180,E1 -19391.282,E2 -19391.282} C_VEL
LIN {X 0,Y 274.424,Z 224.25,A -85,B 0,C 180,E1 -19393.011,E2 -19393.011} C_VEL
LIN {X 0,Y 266.766,Z 210.838,A -85,B 0,C 180,E1 -19395.093,E2 -19395.093} C_VEL
LIN {X 0,Y 259.807,Z 199.919,A -85,B 0,C 180,E1 -19397.117,E2 -19397.117} C_VEL
LIN {X 0,Y 252.301,Z 189.182,A -85,B 0,C 180,E1 -19399.479,E2 -19399.479} C_VEL
LIN {X 0,Y 247.354,Z 182.582,A -85,B 0,C 180,E1 -19401.181,E2 -19401.181} C_VEL
LIN {X 0,Y 244.465,Z 176.654,A -85,B 0,C 180,E1 -19403.429,E2 -19403.429} C_VEL
LIN {X 0,Y 243.397,Z 175.229,A -85,B 0,C 180,E1 -19404.123,E2 -19404.123} C_VEL
LIN {X 0,Y 241.384,Z 173.594,A -85,B 0,C 180,E1 -19405.237,E2 -19405.237} C_VEL
LIN {X 0,Y 238.83,Z 172.92,A -85,B 0,C 180,E1 -19406.367,E2 -19406.367} C_VEL
LIN {X 0,Y 235.716,Z 172.805,A -85,B 0,C 180,E1 -19407.818,E2 -19407.818} C_VEL
LIN {X 0,Y 234.932,Z 172.832,A -85,B 0,C 180,E1 -19408.769,E2 -19408.769} C_VEL
LIN {X 0,Y 234.963,Z 172.834,A -85,B 0,C 180,E1 -19413.342,E2 -19413.342} C_VEL
LIN {X 0,Y 234.984,Z 172.84,A -85,B 0,C 180,E1 -19417.989,E2 -19417.989} C_VEL
LIN {X 0,Y 235.087,Z 172.819,A -85,B 0,C 180,E1 -19423.059,E2 -19423.059} C_VEL
LIN {X 0,Y 235.108,Z 172.798,A -85,B 0,C 180,E1 -19427.921,E2 -19427.921} C_VEL
LIN {X 0,Y 235.38,Z 172.778,A -85,B 0,C 180,E1 -19431.414,E2 -19431.414} C_VEL
LIN {X 0,Y 235.396,Z 172.757,A -85,B 0,C 180,E1 -19433.141,E2 -19433.141} C_VEL
LIN {X 0,Y 235.587,Z 172.747,A -85,B 0,C 180,E1 -19438.29,E2 -19438.29} C_VEL
LIN {X 0,Y 235.587,Z 172.741,A -85,B 0,C 180,E1 -19441.709,E2 -19441.709} C_VEL
LIN {X 0,Y 235.394,Z 172.754,A -85,B 0,C 180,E1 -19446.859,E2 -19446.859} C_VEL
LIN {X 0,Y 235.228,Z 172.803,A -85,B 0,C 180,E1 -19450.327,E2 -19450.327} C_VEL
LIN {X 0,Y 235.103,Z 172.817,A -85,B 0,C 180,E1 -19455.607,E2 -19455.607} C_VEL
LIN {X 0,Y 234.999,Z 172.807,A -85,B 0,C 180,E1 -19459.206,E2 -19459.206} C_VEL
LIN {X 0,Y 234.951,Z 172.83,A -85,B 0,C 180,E1 -19462.884,E2 -19462.884} C_VEL
LIN {X 0,Y 234.959,Z 172.838,A -85,B 0,C 180,E1 -19466.658,E2 -19466.658} C_VEL
LIN {X 0,Y 234.906,Z 172.831,A -85,B 0,C 180,E1 -19470.404,E2 -19470.404} C_VEL
LIN {X 0,Y 235.499,Z 174.93,A -85,B 0,C 180,E1 -19470.983,E2 -19470.983} C_VEL
LIN {X 0,Y 237.565,Z 177.533,A -85,B 0,C 180,E1 -19472.174,E2 -19472.174} C_VEL
LIN {X 0,Y 238.17,Z 177.955,A -85,B 0,C 180,E1 -19472.46,E2 -19472.46} C_VEL
LIN {X 0,Y 239.078,Z 179.983,A -85,B 0,C 180,E1 -19473.074,E2 -19473.074} C_VEL
LIN {X 0,Y 242.477,Z 184.994,A -85,B 0,C 180,E1 -19474.92,E2 -19474.92} C_VEL
LIN {X 0,Y 247.113,Z 191.795,A -85,B 0,C 180,E1 -19477.223,E2 -19477.223} C_VEL
LIN {X 0,Y 252.59,Z 200.77,A -85,B 0,C 180,E1 -19479.788,E2 -19479.788} C_VEL
LIN {X 0,Y 255.045,Z 207.626,A -85,B 0,C 180,E1 -19481.14,E2 -19481.14} C_VEL
LIN {X 0,Y 261.095,Z 221.757,A -85,B 0,C 180,E1 -19483.168,E2 -19483.168} C_VEL
LIN {X 0,Y 269.09,Z 241.325,A -85,B 0,C 180,E1 -19485.64,E2 -19485.64} C_VEL
LIN {X 0,Y 270.133,Z 243.974,A -85,B 0,C 180,E1 -19485.948,E2 -19485.948} C_VEL
LIN {X 0,Y 273.207,Z 286.586,A -85,B 0,C 180,E1 -19488.038,E2 -19488.038} C_VEL
LIN {X 0,Y 268.372,Z 382.289,A -85,B 0,C 180,E1 -19490.458,E2 -19490.458} C_VEL
LIN {X 0,Y 266.841,Z 397.695,A -85,B 0,C 180,E1 -19491.04,E2 -19491.04} C_VEL
LIN {X 0,Y 264.571,Z 412.592,A -85,B 0,C 180,E1 -19491.861,E2 -19491.861} C_VEL
LIN {X 0,Y 261.94,Z 426.079,A -85,B 0,C 180,E1 -19492.868,E2 -19492.868} C_VEL
LIN {X 0,Y 258.535,Z 440.285,A -85,B 0,C 180,E1 -19494.238,E2 -19494.238} C_VEL
LIN {X 0,Y 254.993,Z 453.55,A -85,B 0,C 180,E1 -19495.89,E2 -19495.89} C_VEL
LIN {X 0,Y 251.094,Z 466.34,A -85,B 0,C 180,E1 -19497.876,E2 -19497.876} C_VEL
LIN {X 0,Y 247.809,Z 476.385,A -85,B 0,C 180,E1 -19499.778,E2 -19499.778} C_VEL
LIN {X 0,Y 244.392,Z 486.658,A -85,B 0,C 180,E1 -19502.143,E2 -19502.143} C_VEL
LIN {X 0,Y 240.87,Z 497.129,A -85,B 0,C 180,E1 -19505.126,E2 -19505.126} C_VEL
LIN {X 0,Y 237.866,Z 506.143,A -85,B 0,C 180,E1 -19508.329,E2 -19508.329} C_VEL
LIN {X 0,Y 235.492,Z 513.795,A -85,B 0,C 180,E1 -19511.741,E2 -19511.741} C_VEL
LIN {X 0,Y 233.993,Z 519.907,A -85,B 0,C 180,E1 -19515.211,E2 -19515.211} C_VEL
LIN {X 0,Y 233.19,Z 524.621,A -85,B 0,C 180,E1 -19518.705,E2 -19518.705} C_VEL
LIN {X 0,Y 233.086,Z 527.263,A -85,B 0,C 180,E1 -19521.331,E2 -19521.331} C_VEL
LIN {X 0,Y 233.332,Z 529.746,A -85,B 0,C 180,E1 -19524.818,E2 -19524.818} C_VEL
LIN {X 0,Y 233.644,Z 531.006,A -85,B 0,C 180,E1 -19528.278,E2 -19528.278} C_VEL
LIN {X 0,Y 233.804,Z 531.18,A -85,B 0,C 180,E1 -19530.002,E2 -19530.002} C_VEL
LIN {X 0,Y 233.645,Z 531.004,A -85,B 0,C 180,E1 -19531.726,E2 -19531.726} C_VEL
LIN {X 0,Y 233.362,Z 529.733,A -85,B 0,C 180,E1 -19535.186,E2 -19535.186} C_VEL
LIN {X 0,Y 233.141,Z 527.236,A -85,B 0,C 180,E1 -19538.671,E2 -19538.671} C_VEL
LIN {X 0,Y 233.357,Z 523.488,A -85,B 0,C 180,E1 -19542.172,E2 -19542.172} C_VEL
LIN {X 0,Y 234.306,Z 518.43,A -85,B 0,C 180,E1 -19545.664,E2 -19545.664} C_VEL
LIN {X 0,Y 236.008,Z 511.938,A -85,B 0,C 180,E1 -19549.123,E2 -19549.123} C_VEL
LIN {X 0,Y 238.628,Z 503.836,A -85,B 0,C 180,E1 -19552.514,E2 -19552.514} C_VEL
LIN {X 0,Y 241.521,Z 494.754,A -85,B 0,C 180,E1 -19555.57,E2 -19555.57} C_VEL
LIN {X 0,Y 242.85,Z 491.371,A -85,B 0,C 180,E1 -19556.654,E2 -19556.654} C_VEL
LIN {X 0,Y 247.633,Z 483.795,A -85,B 0,C 180,E1 -19559.781,E2 -19559.781} C_VEL
LIN {X 0,Y 253.401,Z 474.83,A -85,B 0,C 180,E1 -19562.742,E2 -19562.742} C_VEL
LIN {X 0,Y 259.452,Z 465.672,A -85,B 0,C 180,E1 -19565.145,E2 -19565.145} C_VEL
LIN {X 0,Y 266.097,Z 455.105,A -85,B 0,C 180,E1 -19567.408,E2 -19567.408} C_VEL
LIN {X 0,Y 273.487,Z 442.776,A -85,B 0,C 180,E1 -19569.498,E2 -19569.498} C_VEL
LIN {X 0,Y 280.204,Z 430.82,A -85,B 0,C 180,E1 -19571.092,E2 -19571.092} C_VEL
LIN {X 0,Y 287.734,Z 416.164,A -85,B 0,C 180,E1 -19572.604,E2 -19572.604} C_VEL
LIN {X 0,Y 294.54,Z 401.156,A -85,B 0,C 180,E1 -19573.788,E2 -19573.788} C_VEL
LIN {X 0,Y 300.059,Z 387.307,A -85,B 0,C 180,E1 -19574.643,E2 -19574.643} C_VEL
LIN {X 0,Y 305.705,Z 370.209,A -85,B 0,C 180,E1 -19575.455,E2 -19575.455} C_VEL
LIN {X 0,Y 323.205,Z 303.407,A -85,B 0,C 180,E1 -19578.091,E2 -19578.091} C_VEL
LIN {X 0,Y 323.194,Z 303.381,A -85,B 0,C 180,E1 -19578.406,E2 -19578.406} C_VEL
LIN {X 0,Y 312.286,Z 342.814,A -85,B 0,C 180,E1 -19580.157,E2 -19580.157} C_VEL
LIN {X 0,Y 307.633,Z 359.904,A -85,B 0,C 180,E1 -19581.079,E2 -19581.079} C_VEL
LIN {X 0,Y 302.825,Z 374.527,A -85,B 0,C 180,E1 -19582.131,E2 -19582.131} C_VEL
LIN {X 0,Y 297.972,Z 386.664,A -85,B 0,C 180,E1 -19583.238,E2 -19583.238} C_VEL
LIN {X 0,Y 291.924,Z 399.69,A -85,B 0,C 180,E1 -19584.705,E2 -19584.705} C_VEL
LIN {X 0,Y 285.667,Z 411.387,A -85,B 0,C 180,E1 -19586.389,E2 -19586.389} C_VEL
LIN {X 0,Y 278.729,Z 422.721,A -85,B 0,C 180,E1 -19588.453,E2 -19588.453} C_VEL
LIN {X 0,Y 271.41,Z 433.232,A -85,B 0,C 180,E1 -19590.954,E2 -19590.954} C_VEL
LIN {X 0,Y 265.6,Z 440.558,A -85,B 0,C 180,E1 -19593.267,E2 -19593.267} C_VEL
LIN {X 0,Y 260.938,Z 445.796,A -85,B 0,C 180,E1 -19595.325,E2 -19595.325} C_VEL
LIN {X 0,Y 255.234,Z 451.284,A -85,B 0,C 180,E1 -19598.178,E2 -19598.178} C_VEL
LIN {X 0,Y 251.46,Z 454.3,A -85,B 0,C 180,E1 -19600.404,E2 -19600.404} C_VEL
LIN {X 0,Y 246.937,Z 457.034,A -85,B 0,C 180,E1 -19603.465,E2 -19603.465} C_VEL
LIN {X 0,Y 243.19,Z 458.249,A -85,B 0,C 180,E1 -19606.633,E2 -19606.633} C_VEL
LIN {X 0,Y 241.483,Z 458.302,A -85,B 0,C 180,E1 -19608.245,E2 -19608.245} C_VEL
LIN {X 0,Y 238.91,Z 457.202,A -85,B 0,C 180,E1 -19611.542,E2 -19611.542} C_VEL
LIN {X 0,Y 237.974,Z 456.074,A -85,B 0,C 180,E1 -19613.216,E2 -19613.216} C_VEL
LIN {X 0,Y 237.006,Z 454.589,A -85,B 0,C 180,E1 -19614.896,E2 -19614.896} C_VEL
LIN {X 0,Y 236.001,Z 451.575,A -85,B 0,C 180,E1 -19617.44,E2 -19617.44} C_VEL
LIN {X 0,Y 235.157,Z 447.621,A -85,B 0,C 180,E1 -19620,E2 -19620} C_VEL
LIN {X 0,Y 234.928,Z 442.635,A -85,B 0,C 180,E1 -19622.572,E2 -19622.572} C_VEL
LIN {X 0,Y 234.846,Z 435.369,A -85,B 0,C 180,E1 -19625.582,E2 -19625.582} C_VEL
LIN {X 0,Y 235.244,Z 427.73,A -85,B 0,C 180,E1 -19628.158,E2 -19628.158} C_VEL
LIN {X 0,Y 235.704,Z 418.496,A -85,B 0,C 180,E1 -19630.74,E2 -19630.74} C_VEL
LIN {X 0,Y 236.532,Z 407.303,A -85,B 0,C 180,E1 -19633.313,E2 -19633.313} C_VEL
LIN {X 0,Y 237.379,Z 396.058,A -85,B 0,C 180,E1 -19635.454,E2 -19635.454} C_VEL
LIN {X 0,Y 238.454,Z 382.344,A -85,B 0,C 180,E1 -19637.584,E2 -19637.584} C_VEL
LIN {X 0,Y 239.494,Z 369.044,A -85,B 0,C 180,E1 -19639.259,E2 -19639.259} C_VEL
LIN {X 0,Y 240.271,Z 354.995,A -85,B 0,C 180,E1 -19640.661,E2 -19640.661} C_VEL
LIN {X 0,Y 241.017,Z 339.83,A -85,B 0,C 180,E1 -19641.826,E2 -19641.826} C_VEL
LIN {X 0,Y 241.868,Z 319.3,A -85,B 0,C 180,E1 -19642.927,E2 -19642.927} C_VEL
LIN {X 0,Y 246.182,Z 239.576,A -85,B 0,C 180,E1 -19646.73,E2 -19646.73} C_VEL
LIN {X 0,Y 243.105,Z 211.866,A -85,B 0,C 180,E1 -19648.319,E2 -19648.319} C_VEL
LIN {X 0,Y 242.795,Z 207.815,A -85,B 0,C 180,E1 -19648.589,E2 -19648.589} C_VEL
LIN {X 0,Y 240.721,Z 197.758,A -85,B 0,C 180,E1 -19651.704,E2 -19651.704} C_VEL
LIN {X 0,Y 237.976,Z 185.328,A -85,B 0,C 180,E1 -19655.74,E2 -19655.74} C_VEL
LIN {X 0,Y 237.747,Z 184.35,A -85,B 0,C 180,E1 -19656.069,E2 -19656.069} C_VEL
LIN {X 0,Y 238.849,Z 185.899,A -85,B 0,C 180,E1 -19656.537,E2 -19656.537} C_VEL
LIN {X 0,Y 242.675,Z 186.785,A -85,B 0,C 180,E1 -19657.802,E2 -19657.802} C_VEL
LIN {X 0,Y 244.847,Z 189.119,A -85,B 0,C 180,E1 -19658.573,E2 -19658.573} C_VEL
LIN {X 0,Y 252.61,Z 199.959,A -85,B 0,C 180,E1 -19661.233,E2 -19661.233} C_VEL
LIN {X 0,Y 259.458,Z 210.348,A -85,B 0,C 180,E1 -19663.374,E2 -19663.374} C_VEL
LIN {X 0,Y 267.024,Z 223.078,A -85,B 0,C 180,E1 -19665.571,E2 -19665.571} C_VEL
LIN {X 0,Y 274.054,Z 236.721,A -85,B 0,C 180,E1 -19667.501,E2 -19667.501} C_VEL
LIN {X 0,Y 275.835,Z 240.453,A -85,B 0,C 180,E1 -19667.974,E2 -19667.974} C_VEL
LIN {X 0,Y 270.308,Z 348.912,A -85,B 0,C 180,E1 -19670.731,E2 -19670.731} C_VEL
LIN {X 0,Y 268.952,Z 364.161,A -85,B 0,C 180,E1 -19671.38,E2 -19671.38} C_VEL
LIN {X 0,Y 267.276,Z 378.181,A -85,B 0,C 180,E1 -19672.266,E2 -19672.266} C_VEL
LIN {X 0,Y 265.155,Z 391.69,A -85,B 0,C 180,E1 -19673.388,E2 -19673.388} C_VEL
LIN {X 0,Y 262.311,Z 405.502,A -85,B 0,C 180,E1 -19674.825,E2 -19674.825} C_VEL
LIN {X 0,Y 259.232,Z 418.113,A -85,B 0,C 180,E1 -19676.467,E2 -19676.467} C_VEL
LIN {X 0,Y 255.843,Z 429.778,A -85,B 0,C 180,E1 -19678.305,E2 -19678.305} C_VEL
LIN {X 0,Y 252.55,Z 440.557,A -85,B 0,C 180,E1 -19680.397,E2 -19680.397} C_VEL
LIN {X 0,Y 249.252,Z 450.462,A -85,B 0,C 180,E1 -19682.728,E2 -19682.728} C_VEL
LIN {X 0,Y 245.683,Z 460.131,A -85,B 0,C 180,E1 -19685.492,E2 -19685.492} C_VEL
LIN {X 0,Y 242.662,Z 468.13,A -85,B 0,C 180,E1 -19688.328,E2 -19688.328} C_VEL
LIN {X 0,Y 240.035,Z 474.742,A -85,B 0,C 180,E1 -19691.21,E2 -19691.21} C_VEL
LIN {X 0,Y 237.751,Z 480.837,A -85,B 0,C 180,E1 -19694.569,E2 -19694.569} C_VEL
LIN {X 0,Y 236.024,Z 485.54,A -85,B 0,C 180,E1 -19697.967,E2 -19697.967} C_VEL
LIN {X 0,Y 234.827,Z 488.98,A -85,B 0,C 180,E1 -19701.392,E2 -19701.392} C_VEL
LIN {X 0,Y 234.123,Z 491.24,A -85,B 0,C 180,E1 -19704.831,E2 -19704.831} C_VEL
LIN {X 0,Y 233.777,Z 492.386,A -85,B 0,C 180,E1 -19708.275,E2 -19708.275} C_VEL
LIN {X 0,Y 233.776,Z 492.397,A -85,B 0,C 180,E1 -19711.721,E2 -19711.721} C_VEL
LIN {X 0,Y 234.108,Z 491.297,A -85,B 0,C 180,E1 -19715.165,E2 -19715.165} C_VEL
LIN {X 0,Y 234.824,Z 489.085,A -85,B 0,C 180,E1 -19718.604,E2 -19718.604} C_VEL
LIN {X 0,Y 236,Z 485.704,A -85,B 0,C 180,E1 -19722.03,E2 -19722.03} C_VEL
LIN {X 0,Y 237.701,Z 481.058,A -85,B 0,C 180,E1 -19725.43,E2 -19725.43} C_VEL
LIN {X 0,Y 239.981,Z 475.013,A -85,B 0,C 180,E1 -19728.79,E2 -19728.79} C_VEL
LIN {X 0,Y 242.576,Z 468.462,A -85,B 0,C 180,E1 -19731.676,E2 -19731.676} C_VEL
LIN {X 0,Y 245.61,Z 460.514,A -85,B 0,C 180,E1 -19734.511,E2 -19734.511} C_VEL
LIN {X 0,Y 249.151,Z 450.93,A -85,B 0,C 180,E1 -19737.28,E2 -19737.28} C_VEL
LIN {X 0,Y 252.413,Z 441.097,A -85,B 0,C 180,E1 -19739.616,E2 -19739.616} C_VEL
LIN {X 0,Y 255.759,Z 430.422,A -85,B 0,C 180,E1 -19741.702,E2 -19741.702} C_VEL
LIN {X 0,Y 259.093,Z 418.89,A -85,B 0,C 180,E1 -19743.548,E2 -19743.548} C_VEL
LIN {X 0,Y 262.23,Z 406.428,A -85,B 0,C 180,E1 -19745.182,E2 -19745.182} C_VEL
LIN {X 0,Y 265.046,Z 392.85,A -85,B 0,C 180,E1 -19746.625,E2 -19746.625} C_VEL
LIN {X 0,Y 267.352,Z 378.391,A -85,B 0,C 180,E1 -19747.842,E2 -19747.842} C_VEL
LIN {X 0,Y 269.178,Z 363.805,A -85,B 0,C 180,E1 -19748.746,E2 -19748.746} C_VEL
LIN {X 0,Y 270.472,Z 348.094,A -85,B 0,C 180,E1 -19749.416,E2 -19749.416} C_VEL
LIN {X 0,Y 276.002,Z 240.647,A -85,B 0,C 180,E1 -19752.13,E2 -19752.13} C_VEL
LIN {X 0,Y 269.79,Z 228.156,A -85,B 0,C 180,E1 -19753.808,E2 -19753.808} C_VEL
LIN {X 0,Y 262.601,Z 215.444,A -85,B 0,C 180,E1 -19755.848,E2 -19755.848} C_VEL
LIN {X 0,Y 255.984,Z 204.909,A -85,B 0,C 180,E1 -19757.854,E2 -19757.854} C_VEL
LIN {X 0,Y 248.618,Z 194.213,A -85,B 0,C 180,E1 -19760.273,E2 -19760.273} C_VEL
LIN {X 0,Y 241.958,Z 185.34,A -85,B 0,C 180,E1 -19762.671,E2 -19762.671} C_VEL
LIN {X 0,Y 240.252,Z 182.936,A -85,B 0,C 180,E1 -19763.447,E2 -19763.447} C_VEL
LIN {X 0,Y 237.865,Z 178.597,A -85,B 0,C 180,E1 -19765.336,E2 -19765.336} C_VEL
LIN {X 0,Y 237.454,Z 177.393,A -85,B 0,C 180,E1 -19765.781,E2 -19765.781} C_VEL
LIN {X 0,Y 235.238,Z 174.184,A -85,B 0,C 180,E1 -19767.468,E2 -19767.468} C_VEL
LIN {X 0,Y 234.924,Z 172.845,A -85,B 0,C 180,E1 -19767.989,E2 -19767.989} C_VEL
LIN {X 0,Y 234.932,Z 172.832,A -85,B 0,C 180,E1 -19768.769,E2 -19768.769} C_VEL
LIN {X 0,Y 234.247,Z 172.916,A -85,B 0,C 180,E1 -19770.2,E2 -19770.2} C_VEL
LIN {X 0,Y 231.426,Z 173.284,A -85,B 0,C 180,E1 -19772.538,E2 -19772.538} C_VEL
LIN {X 0,Y 229.034,Z 173.567,A -85,B 0,C 180,E1 -19774.443,E2 -19774.443} C_VEL
LIN {X 0,Y 227.996,Z 173.688,A -85,B 0,C 180,E1 -19775.921,E2 -19775.921} C_VEL
LIN {X 0,Y 227.903,Z 173.702,A -85,B 0,C 180,E1 -19776.421,E2 -19776.421} C_VEL
LIN {X 0,Y 227.933,Z 173.693,A -85,B 0,C 180,E1 -19780.173,E2 -19780.173} C_VEL
LIN {X 0,Y 228.048,Z 173.704,A -85,B 0,C 180,E1 -19783.897,E2 -19783.897} C_VEL
LIN {X 0,Y 228.065,Z 173.672,A -85,B 0,C 180,E1 -19787.543,E2 -19787.543} C_VEL
LIN {X 0,Y 228.315,Z 173.662,A -85,B 0,C 180,E1 -19791.146,E2 -19791.146} C_VEL
LIN {X 0,Y 228.348,Z 173.635,A -85,B 0,C 180,E1 -19792.928,E2 -19792.928} C_VEL
LIN {X 0,Y 228.546,Z 173.624,A -85,B 0,C 180,E1 -19798.238,E2 -19798.238} C_VEL
LIN {X 0,Y 228.546,Z 173.618,A -85,B 0,C 180,E1 -19801.762,E2 -19801.762} C_VEL
LIN {X 0,Y 228.345,Z 173.631,A -85,B 0,C 180,E1 -19807.072,E2 -19807.072} C_VEL
LIN {X 0,Y 228.149,Z 173.681,A -85,B 0,C 180,E1 -19810.651,E2 -19810.651} C_VEL
LIN {X 0,Y 228.054,Z 173.674,A -85,B 0,C 180,E1 -19814.273,E2 -19814.273} C_VEL
LIN {X 0,Y 227.993,Z 173.683,A -85,B 0,C 180,E1 -19817.954,E2 -19817.954} C_VEL
LIN {X 0,Y 227.921,Z 173.714,A -85,B 0,C 180,E1 -19822.33,E2 -19822.33} C_VEL
LIN {X 0,Y 227.897,Z 173.722,A -85,B 0,C 180,E1 -19826.987,E2 -19826.987} C_VEL
LIN {X 0,Y 227.914,Z 173.876,A -85,B 0,C 180,E1 -19827.48,E2 -19827.48} C_VEL
LIN {X 0,Y 228.885,Z 176.572,A -85,B 0,C 180,E1 -19828.42,E2 -19828.42} C_VEL
LIN {X 0,Y 230.933,Z 178.688,A -85,B 0,C 180,E1 -19829.694,E2 -19829.694} C_VEL
LIN {X 0,Y 232.659,Z 181.814,A -85,B 0,C 180,E1 -19830.899,E2 -19830.899} C_VEL
LIN {X 0,Y 234.733,Z 184.297,A -85,B 0,C 180,E1 -19832.103,E2 -19832.103} C_VEL
LIN {X 0,Y 241.817,Z 195.361,A -85,B 0,C 180,E1 -19836.053,E2 -19836.053} C_VEL
LIN {X 0,Y 248.307,Z 205.972,A -85,B 0,C 180,E1 -19839.259,E2 -19839.259} C_VEL
LIN {X 0,Y 253.743,Z 218.576,A -85,B 0,C 180,E1 -19841.265,E2 -19841.265} C_VEL
LIN {X 0,Y 259.238,Z 231.851,A -85,B 0,C 180,E1 -19843.134,E2 -19843.134} C_VEL
LIN {X 0,Y 265.149,Z 247.046,A -85,B 0,C 180,E1 -19845.027,E2 -19845.027} C_VEL
LIN {X 0,Y 267.839,Z 287.152,A -85,B 0,C 180,E1 -19847.034,E2 -19847.034} C_VEL
LIN {X 0,Y 264.596,Z 352.296,A -85,B 0,C 180,E1 -19848.712,E2 -19848.712} C_VEL
LIN {X 0,Y 262.619,Z 385.959,A -85,B 0,C 180,E1 -19849.603,E2 -19849.603} C_VEL
LIN {X 0,Y 260.769,Z 401.475,A -85,B 0,C 180,E1 -19850.268,E2 -19850.268} C_VEL
LIN {X 0,Y 258.365,Z 415.84,A -85,B 0,C 180,E1 -19851.149,E2 -19851.149} C_VEL
LIN {X 0,Y 255.407,Z 429.453,A -85,B 0,C 180,E1 -19852.251,E2 -19852.251} C_VEL
LIN {X 0,Y 251.922,Z 442.865,A -85,B 0,C 180,E1 -19853.645,E2 -19853.645} C_VEL
LIN {X 0,Y 248.413,Z 455.33,A -85,B 0,C 180,E1 -19855.306,E2 -19855.306} C_VEL
LIN {X 0,Y 244.337,Z 467.902,A -85,B 0,C 180,E1 -19857.366,E2 -19857.366} C_VEL
LIN {X 0,Y 241.011,Z 477.596,A -85,B 0,C 180,E1 -19859.318,E2 -19859.318} C_VEL
LIN {X 0,Y 237.51,Z 487.583,A -85,B 0,C 180,E1 -19861.745,E2 -19861.745} C_VEL
LIN {X 0,Y 234.218,Z 496.89,A -85,B 0,C 180,E1 -19864.503,E2 -19864.503} C_VEL
LIN {X 0,Y 231.185,Z 505.551,A -85,B 0,C 180,E1 -19867.669,E2 -19867.669} C_VEL
LIN {X 0,Y 228.666,Z 513.202,A -85,B 0,C 180,E1 -19871.175,E2 -19871.175} C_VEL
LIN {X 0,Y 227.049,Z 519.315,A -85,B 0,C 180,E1 -19874.748,E2 -19874.748} C_VEL
LIN {X 0,Y 226.15,Z 524.028,A -85,B 0,C 180,E1 -19878.349,E2 -19878.349} C_VEL
LIN {X 0,Y 225.984,Z 526.67,A -85,B 0,C 180,E1 -19881.057,E2 -19881.057} C_VEL
LIN {X 0,Y 226.247,Z 529.158,A -85,B 0,C 180,E1 -19884.655,E2 -19884.655} C_VEL
LIN {X 0,Y 226.546,Z 530.42,A -85,B 0,C 180,E1 -19888.225,E2 -19888.225} C_VEL
LIN {X 0,Y 226.745,Z 530.596,A -85,B 0,C 180,E1 -19890.002,E2 -19890.002} C_VEL
LIN {X 0,Y 226.321,Z 529.925,A -85,B 0,C 180,E1 -19893.563,E2 -19893.563} C_VEL
LIN {X 0,Y 226.247,Z 528.635,A -85,B 0,C 180,E1 -19896.267,E2 -19896.267} C_VEL
LIN {X 0,Y 226.056,Z 526.643,A -85,B 0,C 180,E1 -19898.945,E2 -19898.945} C_VEL
LIN {X 0,Y 226.337,Z 522.894,A -85,B 0,C 180,E1 -19902.556,E2 -19902.556} C_VEL
LIN {X 0,Y 227.372,Z 517.834,A -85,B 0,C 180,E1 -19906.154,E2 -19906.154} C_VEL
LIN {X 0,Y 229.226,Z 511.344,A -85,B 0,C 180,E1 -19909.712,E2 -19909.712} C_VEL
LIN {X 0,Y 231.963,Z 503.239,A -85,B 0,C 180,E1 -19913.198,E2 -19913.198} C_VEL
LIN {X 0,Y 234.766,Z 494.935,A -85,B 0,C 180,E1 -19916.093,E2 -19916.093} C_VEL
LIN {X 0,Y 235.673,Z 492.675,A -85,B 0,C 180,E1 -19916.813,E2 -19916.813} C_VEL
LIN {X 0,Y 240.135,Z 486.2,A -85,B 0,C 180,E1 -19919.839,E2 -19919.839} C_VEL
LIN {X 0,Y 246.701,Z 476.975,A -85,B 0,C 180,E1 -19923.259,E2 -19923.259} C_VEL
LIN {X 0,Y 252.826,Z 468.464,A -85,B 0,C 180,E1 -19925.717,E2 -19925.717} C_VEL
LIN {X 0,Y 260.649,Z 457.172,A -85,B 0,C 180,E1 -19928.33,E2 -19928.33} C_VEL
LIN {X 0,Y 268.267,Z 445.599,A -85,B 0,C 180,E1 -19930.423,E2 -19930.423} C_VEL
LIN {X 0,Y 276.144,Z 432.765,A -85,B 0,C 180,E1 -19932.231,E2 -19932.231} C_VEL
LIN {X 0,Y 283.695,Z 419.321,A -85,B 0,C 180,E1 -19933.676,E2 -19933.676} C_VEL
LIN {X 0,Y 290.425,Z 405.963,A -85,B 0,C 180,E1 -19934.815,E2 -19934.815} C_VEL
LIN {X 0,Y 297.496,Z 389.96,A -85,B 0,C 180,E1 -19935.857,E2 -19935.857} C_VEL
LIN {X 0,Y 303.73,Z 372.938,A -85,B 0,C 180,E1 -19936.673,E2 -19936.673} C_VEL
LIN {X 0,Y 309.198,Z 354.24,A -85,B 0,C 180,E1 -19937.443,E2 -19937.443} C_VEL
LIN {X 0,Y 315.003,Z 332.678,A -85,B 0,C 180,E1 -19938.272,E2 -19938.272} C_VEL
LIN {X 0,Y 314.98,Z 332.74,A -85,B 0,C 180,E1 -19938.347,E2 -19938.347} C_VEL
LIN {X 0,Y 307.255,Z 359.738,A -85,B 0,C 180,E1 -19939.693,E2 -19939.693} C_VEL
LIN {X 0,Y 302.317,Z 374.354,A -85,B 0,C 180,E1 -19940.693,E2 -19940.693} C_VEL
LIN {X 0,Y 296.388,Z 388.441,A -85,B 0,C 180,E1 -19941.938,E2 -19941.938} C_VEL
LIN {X 0,Y 290.025,Z 401.183,A -85,B 0,C 180,E1 -19943.365,E2 -19943.365} C_VEL
LIN {X 0,Y 283.943,Z 411.87,A -85,B 0,C 180,E1 -19944.868,E2 -19944.868} C_VEL
LIN {X 0,Y 277.593,Z 421.746,A -85,B 0,C 180,E1 -19946.588,E2 -19946.588} C_VEL
LIN {X 0,Y 270.658,Z 431.352,A -85,B 0,C 180,E1 -19948.713,E2 -19948.713} C_VEL
LIN {X 0,Y 265.071,Z 438.224,A -85,B 0,C 180,E1 -19950.627,E2 -19950.627} C_VEL
LIN {X 0,Y 259.907,Z 444.019,A -85,B 0,C 180,E1 -19952.633,E2 -19952.633} C_VEL
LIN {X 0,Y 253.468,Z 450.224,A -85,B 0,C 180,E1 -19955.424,E2 -19955.424} C_VEL
LIN {X 0,Y 247.71,Z 454.829,A -85,B 0,C 180,E1 -19958.356,E2 -19958.356} C_VEL
LIN {X 0,Y 242.658,Z 457.903,A -85,B 0,C 180,E1 -19961.423,E2 -19961.423} C_VEL
LIN {X 0,Y 238.288,Z 459.48,A -85,B 0,C 180,E1 -19964.607,E2 -19964.607} C_VEL
LIN {X 0,Y 234.661,Z 459.583,A -85,B 0,C 180,E1 -19967.899,E2 -19967.899} C_VEL
LIN {X 0,Y 231.966,Z 458.177,A -85,B 0,C 180,E1 -19971.287,E2 -19971.287} C_VEL
LIN {X 0,Y 230.981,Z 456.9,A -85,B 0,C 180,E1 -19973.01,E2 -19973.01} C_VEL
LIN {X 0,Y 229.611,Z 454.245,A -85,B 0,C 180,E1 -19975.612,E2 -19975.612} C_VEL
LIN {X 0,Y 228.59,Z 450.676,A -85,B 0,C 180,E1 -19978.238,E2 -19978.238} C_VEL
LIN {X 0,Y 228.034,Z 446.132,A -85,B 0,C 180,E1 -19980.883,E2 -19980.883} C_VEL
LIN {X 0,Y 227.752,Z 439.472,A -85,B 0,C 180,E1 -19983.981,E2 -19983.981} C_VEL
LIN {X 0,Y 227.938,Z 431.129,A -85,B 0,C 180,E1 -19987.085,E2 -19987.085} C_VEL
LIN {X 0,Y 228.386,Z 422.126,A -85,B 0,C 180,E1 -19989.811,E2 -19989.811} C_VEL
LIN {X 0,Y 229.092,Z 411.825,A -85,B 0,C 180,E1 -19992.401,E2 -19992.401} C_VEL
LIN {X 0,Y 230.014,Z 400.085,A -85,B 0,C 180,E1 -19994.827,E2 -19994.827} C_VEL
LIN {X 0,Y 230.974,Z 387.158,A -85,B 0,C 180,E1 -19997.03,E2 -19997.03} C_VEL
LIN {X 0,Y 231.971,Z 374.518,A -85,B 0,C 180,E1 -19998.778,E2 -19998.778} C_VEL
LIN {X 0,Y 232.903,Z 360.464,A -85,B 0,C 180,E1 -20000.35,E2 -20000.35} C_VEL
LIN {X 0,Y 233.785,Z 345.273,A -85,B 0,C 180,E1 -20001.666,E2 -20001.666} C_VEL
LIN {X 0,Y 234.394,Z 329.838,A -85,B 0,C 180,E1 -20002.65,E2 -20002.65} C_VEL
LIN {X 0,Y 238.688,Z 250.885,A -85,B 0,C 180,E1 -20006.584,E2 -20006.584} C_VEL
LIN {X 0,Y 239.17,Z 239.018,A -85,B 0,C 180,E1 -20007.172,E2 -20007.172} C_VEL
LIN {X 0,Y 236.466,Z 214.654,A -85,B 0,C 180,E1 -20008.609,E2 -20008.609} C_VEL
LIN {X 0,Y 235.78,Z 208.386,A -85,B 0,C 180,E1 -20008.983,E2 -20008.983} C_VEL
LIN {X 0,Y 232.807,Z 194.495,A -85,B 0,C 180,E1 -20013.431,E2 -20013.431} C_VEL
LIN {X 0,Y 232.162,Z 191.436,A -85,B 0,C 180,E1 -20014.505,E2 -20014.505} C_VEL
LIN {X 0,Y 233.151,Z 192.881,A -85,B 0,C 180,E1 -20014.941,E2 -20014.941} C_VEL
LIN {X 0,Y 237.616,Z 192.976,A -85,B 0,C 180,E1 -20016.485,E2 -20016.485} C_VEL
LIN {X 0,Y 240.833,Z 193.634,A -85,B 0,C 180,E1 -20017.557,E2 -20017.557} C_VEL
LIN {X 0,Y 248.745,Z 204.699,A -85,B 0,C 180,E1 -20020.398,E2 -20020.398} C_VEL
LIN {X 0,Y 255.925,Z 215.887,A -85,B 0,C 180,E1 -20022.743,E2 -20022.743} C_VEL
LIN {X 0,Y 262.8,Z 227.639,A -85,B 0,C 180,E1 -20024.821,E2 -20024.821} C_VEL
LIN {X 0,Y 269.267,Z 240.317,A -85,B 0,C 180,E1 -20026.674,E2 -20026.674} C_VEL
LIN {X 0,Y 270.486,Z 242.961,A -85,B 0,C 180,E1 -20027.016,E2 -20027.016} C_VEL
LIN {X 0,Y 267.695,Z 296.019,A -85,B 0,C 180,E1 -20028.361,E2 -20028.361} C_VEL
LIN {X 0,Y 264.77,Z 350.814,A -85,B 0,C 180,E1 -20029.806,E2 -20029.806} C_VEL
LIN {X 0,Y 263.344,Z 366.1,A -85,B 0,C 180,E1 -20030.498,E2 -20030.498} C_VEL
LIN {X 0,Y 261.513,Z 380.291,A -85,B 0,C 180,E1 -20031.436,E2 -20031.436} C_VEL
LIN {X 0,Y 259.161,Z 394.176,A -85,B 0,C 180,E1 -20032.642,E2 -20032.642} C_VEL
LIN {X 0,Y 256.576,Z 406.075,A -85,B 0,C 180,E1 -20033.918,E2 -20033.918} C_VEL
LIN {X 0,Y 253.379,Z 418.689,A -85,B 0,C 180,E1 -20035.586,E2 -20035.586} C_VEL
LIN {X 0,Y 249.844,Z 430.359,A -85,B 0,C 180,E1 -20037.452,E2 -20037.452} C_VEL
LIN {X 0,Y 246.4,Z 441.141,A -85,B 0,C 180,E1 -20039.582,E2 -20039.582} C_VEL
LIN {X 0,Y 242.986,Z 451.044,A -85,B 0,C 180,E1 -20041.963,E2 -20041.963} C_VEL
LIN {X 0,Y 239.249,Z 460.715,A -85,B 0,C 180,E1 -20044.788,E2 -20044.788} C_VEL
LIN {X 0,Y 236.073,Z 468.716,A -85,B 0,C 180,E1 -20047.691,E2 -20047.691} C_VEL
LIN {X 0,Y 233.332,Z 475.328,A -85,B 0,C 180,E1 -20050.649,E2 -20050.649} C_VEL
LIN {X 0,Y 230.929,Z 481.423,A -85,B 0,C 180,E1 -20054.101,E2 -20054.101} C_VEL
LIN {X 0,Y 229.086,Z 486.128,A -85,B 0,C 180,E1 -20057.597,E2 -20057.597} C_VEL
LIN {X 0,Y 227.819,Z 489.566,A -85,B 0,C 180,E1 -20061.125,E2 -20061.125} C_VEL
LIN {X 0,Y 227.064,Z 491.826,A -85,B 0,C 180,E1 -20064.67,E2 -20064.67} C_VEL
LIN {X 0,Y 226.732,Z 492.969,A -85,B 0,C 180,E1 -20068.221,E2 -20068.221} C_VEL
LIN {X 0,Y 226.731,Z 492.98,A -85,B 0,C 180,E1 -20071.774,E2 -20071.774} C_VEL
LIN {X 0,Y 227.048,Z 491.883,A -85,B 0,C 180,E1 -20075.326,E2 -20075.326} C_VEL
LIN {X 0,Y 227.995,Z 489.209,A -85,B 0,C 180,E1 -20079.457,E2 -20079.457} C_VEL
LIN {X 0,Y 229.455,Z 485.267,A -85,B 0,C 180,E1 -20083.278,E2 -20083.278} C_VEL
LIN {X 0,Y 231.425,Z 480.268,A -85,B 0,C 180,E1 -20086.766,E2 -20086.766} C_VEL
LIN {X 0,Y 234.066,Z 473.84,A -85,B 0,C 180,E1 -20090.197,E2 -20090.197} C_VEL
LIN {X 0,Y 237.149,Z 466.024,A -85,B 0,C 180,E1 -20093.488,E2 -20093.488} C_VEL
LIN {X 0,Y 240.711,Z 457.181,A -85,B 0,C 180,E1 -20096.437,E2 -20096.437} C_VEL
LIN {X 0,Y 244.042,Z 448.367,A -85,B 0,C 180,E1 -20098.838,E2 -20098.838} C_VEL
LIN {X 0,Y 247.636,Z 437.551,A -85,B 0,C 180,E1 -20101.299,E2 -20101.299} C_VEL
LIN {X 0,Y 251.455,Z 425.481,A -85,B 0,C 180,E1 -20103.501,E2 -20103.501} C_VEL
LIN {X 0,Y 255.001,Z 412.833,A -85,B 0,C 180,E1 -20105.361,E2 -20105.361} C_VEL
LIN {X 0,Y 257.931,Z 400.574,A -85,B 0,C 180,E1 -20106.827,E2 -20106.827} C_VEL
LIN {X 0,Y 260.692,Z 386.335,A -85,B 0,C 180,E1 -20108.194,E2 -20108.194} C_VEL
LIN {X 0,Y 262.835,Z 371.325,A -85,B 0,C 180,E1 -20109.312,E2 -20109.312} C_VEL
LIN {X 0,Y 264.502,Z 355.863,A -85,B 0,C 180,E1 -20110.113,E2 -20110.113} C_VEL
LIN {X 0,Y 265.589,Z 339.111,A -85,B 0,C 180,E1 -20110.661,E2 -20110.661} C_VEL
LIN {X 0,Y 270.658,Z 243.142,A -85,B 0,C 180,E1 -20113.088,E2 -20113.088} C_VEL
LIN {X 0,Y 265.431,Z 232.547,A -85,B 0,C 180,E1 -20114.566,E2 -20114.566} C_VEL
LIN {X 0,Y 258.8,Z 220.588,A -85,B 0,C 180,E1 -20116.53,E2 -20116.53} C_VEL
LIN {X 0,Y 252.15,Z 209.804,A -85,B 0,C 180,E1 -20118.632,E2 -20118.632} C_VEL
LIN {X 0,Y 245.158,Z 199.5,A -85,B 0,C 180,E1 -20121.028,E2 -20121.028} C_VEL
LIN {X 0,Y 238.653,Z 190.717,A -85,B 0,C 180,E1 -20123.471,E2 -20123.471} C_VEL
LIN {X 0,Y 234.95,Z 186.071,A -85,B 0,C 180,E1 -20124.974,E2 -20124.974} C_VEL
LIN {X 0,Y 233.454,Z 183.965,A -85,B 0,C 180,E1 -20125.705,E2 -20125.705} C_VEL
LIN {X 0,Y 232.947,Z 182.725,A -85,B 0,C 180,E1 -20126.212,E2 -20126.212} C_VEL
LIN {X 0,Y 228.087,Z 174.641,A -85,B 0,C 180,E1 -20130.462,E2 -20130.462} C_VEL
LIN {X 0,Y 227.909,Z 173.702,A -85,B 0,C 180,E1 -20130.879,E2 -20130.879} C_VEL
LIN {X 0,Y 227.92,Z 173.698,A -85,B 0,C 180,E1 -20134.425,E2 -20134.425} C_VEL
LIN {X 0,Y 227.903,Z 173.702,A -85,B 0,C 180,E1 -20136.421,E2 -20136.421} C_VEL
LIN {X 0,Y 227.228,Z 173.807,A -85,B 0,C 180,E1 -20137.897,E2 -20137.897} C_VEL
LIN {X 0,Y 224.43,Z 174.155,A -85,B 0,C 180,E1 -20140.309,E2 -20140.309} C_VEL
LIN {X 0,Y 222.065,Z 174.446,A -85,B 0,C 180,E1 -20142.275,E2 -20142.275} C_VEL
LIN {X 0,Y 221.05,Z 174.576,A -85,B 0,C 180,E1 -20143.8,E2 -20143.8} C_VEL
LIN {X 0,Y 220.966,Z 174.571,A -85,B 0,C 180,E1 -20144.317,E2 -20144.317} C_VEL
LIN {X 0,Y 221.218,Z 174.555,A -85,B 0,C 180,E1 -20150,E2 -20150} C_VEL
LIN {X 0,Y 221.285,Z 174.516,A -85,B 0,C 180,E1 -20152.701,E2 -20152.701} C_VEL
LIN {X 0,Y 221.504,Z 174.501,A -85,B 0,C 180,E1 -20158.182,E2 -20158.182} C_VEL
LIN {X 0,Y 221.504,Z 174.495,A -85,B 0,C 180,E1 -20161.818,E2 -20161.818} C_VEL
LIN {X 0,Y 221.28,Z 174.511,A -85,B 0,C 180,E1 -20167.299,E2 -20167.299} C_VEL
LIN {X 0,Y 221.097,Z 174.551,A -85,B 0,C 180,E1 -20170.995,E2 -20170.995} C_VEL
LIN {X 0,Y 221.007,Z 174.572,A -85,B 0,C 180,E1 -20176.63,E2 -20176.63} C_VEL
LIN {X 0,Y 220.883,Z 174.574,A -85,B 0,C 180,E1 -20180.487,E2 -20180.487} C_VEL
LIN {X 0,Y 220.863,Z 174.635,A -85,B 0,C 180,E1 -20183.94,E2 -20183.94} C_VEL
LIN {X 0,Y 221.163,Z 175.957,A -85,B 0,C 180,E1 -20184.4,E2 -20184.4} C_VEL
LIN {X 0,Y 222.096,Z 177.741,A -85,B 0,C 180,E1 -20185.289,E2 -20185.289} C_VEL
LIN {X 0,Y 224.545,Z 180.221,A -85,B 0,C 180,E1 -20187.037,E2 -20187.037} C_VEL
LIN {X 0,Y 225.456,Z 182.392,A -85,B 0,C 180,E1 -20187.877,E2 -20187.877} C_VEL
LIN {X 0,Y 227.957,Z 185.516,A -85,B 0,C 180,E1 -20189.557,E2 -20189.557} C_VEL
LIN {X 0,Y 229.126,Z 187.609,A -85,B 0,C 180,E1 -20190.405,E2 -20190.405} C_VEL
LIN {X 0,Y 231.327,Z 190.462,A -85,B 0,C 180,E1 -20191.72,E2 -20191.72} C_VEL
LIN {X 0,Y 238.118,Z 201.208,A -85,B 0,C 180,E1 -20195.66,E2 -20195.66} C_VEL
LIN {X 0,Y 241.644,Z 206.82,A -85,B 0,C 180,E1 -20197.381,E2 -20197.381} C_VEL
LIN {X 0,Y 245.108,Z 211.987,A -85,B 0,C 180,E1 -20198.648,E2 -20198.648} C_VEL
LIN {X 0,Y 252.134,Z 228.886,A -85,B 0,C 180,E1 -20201.286,E2 -20201.286} C_VEL
LIN {X 0,Y 260.186,Z 249.572,A -85,B 0,C 180,E1 -20204.04,E2 -20204.04} C_VEL
LIN {X 0,Y 262.658,Z 289.002,A -85,B 0,C 180,E1 -20206.057,E2 -20206.057} C_VEL
LIN {X 0,Y 257.367,Z 384.206,A -85,B 0,C 180,E1 -20208.535,E2 -20208.535} C_VEL
LIN {X 0,Y 255.454,Z 400.173,A -85,B 0,C 180,E1 -20209.204,E2 -20209.204} C_VEL
LIN {X 0,Y 252.863,Z 415.286,A -85,B 0,C 180,E1 -20210.137,E2 -20210.137} C_VEL
LIN {X 0,Y 249.823,Z 428.892,A -85,B 0,C 180,E1 -20211.252,E2 -20211.252} C_VEL
LIN {X 0,Y 246.219,Z 442.295,A -85,B 0,C 180,E1 -20212.662,E2 -20212.662} C_VEL
LIN {X 0,Y 242.603,Z 454.608,A -85,B 0,C 180,E1 -20214.322,E2 -20214.322} C_VEL
LIN {X 0,Y 238.361,Z 467.324,A -85,B 0,C 180,E1 -20216.441,E2 -20216.441} C_VEL
LIN {X 0,Y 234.851,Z 477.01,A -85,B 0,C 180,E1 -20218.422,E2 -20218.422} C_VEL
LIN {X 0,Y 231.194,Z 486.995,A -85,B 0,C 180,E1 -20220.9,E2 -20220.9} C_VEL
LIN {X 0,Y 227.763,Z 496.065,A -85,B 0,C 180,E1 -20223.636,E2 -20223.636} C_VEL
LIN {X 0,Y 224.552,Z 504.961,A -85,B 0,C 180,E1 -20226.972,E2 -20226.972} C_VEL
LIN {X 0,Y 221.842,Z 512.608,A -85,B 0,C 180,E1 -20230.573,E2 -20230.573} C_VEL
LIN {X 0,Y 220.119,Z 518.723,A -85,B 0,C 180,E1 -20234.256,E2 -20234.256} C_VEL
LIN {X 0,Y 219.108,Z 523.435,A -85,B 0,C 180,E1 -20237.969,E2 -20237.969} C_VEL
LIN {X 0,Y 218.907,Z 526.078,A -85,B 0,C 180,E1 -20240.765,E2 -20240.765} C_VEL
LIN {X 0,Y 219.163,Z 528.57,A -85,B 0,C 180,E1 -20244.482,E2 -20244.482} C_VEL
LIN {X 0,Y 219.449,Z 529.833,A -85,B 0,C 180,E1 -20248.167,E2 -20248.167} C_VEL
LIN {X 0,Y 219.686,Z 530.013,A -85,B 0,C 180,E1 -20250.002,E2 -20250.002} C_VEL
LIN {X 0,Y 219.243,Z 529.339,A -85,B 0,C 180,E1 -20253.678,E2 -20253.678} C_VEL
LIN {X 0,Y 219.16,Z 528.201,A -85,B 0,C 180,E1 -20256.227,E2 -20256.227} C_VEL
LIN {X 0,Y 218.967,Z 526.05,A -85,B 0,C 180,E1 -20259.237,E2 -20259.237} C_VEL
LIN {X 0,Y 219.328,Z 522.299,A -85,B 0,C 180,E1 -20262.964,E2 -20262.964} C_VEL
LIN {X 0,Y 220.461,Z 517.239,A -85,B 0,C 180,E1 -20266.675,E2 -20266.675} C_VEL
LIN {X 0,Y 222.45,Z 510.749,A -85,B 0,C 180,E1 -20270.339,E2 -20270.339} C_VEL
LIN {X 0,Y 225.365,Z 502.645,A -85,B 0,C 180,E1 -20273.919,E2 -20273.919} C_VEL
LIN {X 0,Y 228.69,Z 493.514,A -85,B 0,C 180,E1 -20277.148,E2 -20277.148} C_VEL
LIN {X 0,Y 234.001,Z 486.567,A -85,B 0,C 180,E1 -20280.705,E2 -20280.705} C_VEL
LIN {X 0,Y 240.858,Z 477.809,A -85,B 0,C 180,E1 -20284.175,E2 -20284.175} C_VEL
LIN {X 0,Y 245.327,Z 472.216,A -85,B 0,C 180,E1 -20285.966,E2 -20285.966} C_VEL
LIN {X 0,Y 254.226,Z 460.646,A -85,B 0,C 180,E1 -20288.972,E2 -20288.972} C_VEL
LIN {X 0,Y 263.116,Z 448.338,A -85,B 0,C 180,E1 -20291.386,E2 -20291.386} C_VEL
LIN {X 0,Y 271.806,Z 435.396,A -85,B 0,C 180,E1 -20293.319,E2 -20293.319} C_VEL
LIN {X 0,Y 279.553,Z 422.86,A -85,B 0,C 180,E1 -20294.745,E2 -20294.745} C_VEL
LIN {X 0,Y 287.156,Z 409.199,A -85,B 0,C 180,E1 -20295.969,E2 -20295.969} C_VEL
LIN {X 0,Y 295.102,Z 392.693,A -85,B 0,C 180,E1 -20297.084,E2 -20297.084} C_VEL
LIN {X 0,Y 301.925,Z 376.048,A -85,B 0,C 180,E1 -20297.901,E2 -20297.901} C_VEL
LIN {X 0,Y 305.604,Z 365.195,A -85,B 0,C 180,E1 -20298.35,E2 -20298.35} C_VEL
LIN {X 0,Y 305.444,Z 365.549,A -85,B 0,C 180,E1 -20298.66,E2 -20298.66} C_VEL
LIN {X 0,Y 300.23,Z 379.173,A -85,B 0,C 180,E1 -20299.634,E2 -20299.634} C_VEL
LIN {X 0,Y 293.846,Z 392.93,A -85,B 0,C 180,E1 -20300.89,E2 -20300.89} C_VEL
LIN {X 0,Y 286.031,Z 407.054,A -85,B 0,C 180,E1 -20302.546,E2 -20302.546} C_VEL
LIN {X 0,Y 278.022,Z 419.369,A -85,B 0,C 180,E1 -20304.451,E2 -20304.451} C_VEL
LIN {X 0,Y 270.456,Z 429.537,A -85,B 0,C 180,E1 -20306.482,E2 -20306.482} C_VEL
LIN {X 0,Y 263.596,Z 437.661,A -85,B 0,C 180,E1 -20308.563,E2 -20308.563} C_VEL
LIN {X 0,Y 257.756,Z 443.924,A -85,B 0,C 180,E1 -20310.608,E2 -20310.608} C_VEL
LIN {X 0,Y 250.776,Z 450.425,A -85,B 0,C 180,E1 -20313.359,E2 -20313.359} C_VEL
LIN {X 0,Y 244.374,Z 455.36,A -85,B 0,C 180,E1 -20316.258,E2 -20316.258} C_VEL
LIN {X 0,Y 238.766,Z 458.706,A -85,B 0,C 180,E1 -20319.316,E2 -20319.316} C_VEL
LIN {X 0,Y 233.797,Z 460.651,A -85,B 0,C 180,E1 -20322.506,E2 -20322.506} C_VEL
LIN {X 0,Y 229.714,Z 461.133,A -85,B 0,C 180,E1 -20325.833,E2 -20325.833} C_VEL
LIN {X 0,Y 227.842,Z 460.84,A -85,B 0,C 180,E1 -20327.531,E2 -20327.531} C_VEL
LIN {X 0,Y 225.009,Z 459.051,A -85,B 0,C 180,E1 -20331.015,E2 -20331.015} C_VEL
LIN {X 0,Y 223.991,Z 457.59,A -85,B 0,C 180,E1 -20332.79,E2 -20332.79} C_VEL
LIN {X 0,Y 222.557,Z 454.714,A -85,B 0,C 180,E1 -20335.472,E2 -20335.472} C_VEL
LIN {X 0,Y 221.494,Z 450.915,A -85,B 0,C 180,E1 -20338.182,E2 -20338.182} C_VEL
LIN {X 0,Y 220.929,Z 446.104,A -85,B 0,C 180,E1 -20340.912,E2 -20340.912} C_VEL
LIN {X 0,Y 220.671,Z 439.108,A -85,B 0,C 180,E1 -20344.109,E2 -20344.109} C_VEL
LIN {X 0,Y 220.897,Z 430.384,A -85,B 0,C 180,E1 -20347.312,E2 -20347.312} C_VEL
LIN {X 0,Y 221.386,Z 420.708,A -85,B 0,C 180,E1 -20350.218,E2 -20350.218} C_VEL
LIN {X 0,Y 222.201,Z 409.248,A -85,B 0,C 180,E1 -20353.024,E2 -20353.024} C_VEL
LIN {X 0,Y 223.089,Z 398.072,A -85,B 0,C 180,E1 -20355.298,E2 -20355.298} C_VEL
LIN {X 0,Y 224.161,Z 384.41,A -85,B 0,C 180,E1 -20357.564,E2 -20357.564} C_VEL
LIN {X 0,Y 225.217,Z 371.096,A -85,B 0,C 180,E1 -20359.364,E2 -20359.364} C_VEL
LIN {X 0,Y 226.163,Z 355.319,A -85,B 0,C 180,E1 -20361.04,E2 -20361.04} C_VEL
LIN {X 0,Y 226.938,Z 340.493,A -85,B 0,C 180,E1 -20362.235,E2 -20362.235} C_VEL
LIN {X 0,Y 228.021,Z 315.963,A -85,B 0,C 180,E1 -20363.621,E2 -20363.621} C_VEL
LIN {X 0,Y 232.31,Z 240.607,A -85,B 0,C 180,E1 -20367.505,E2 -20367.505} C_VEL
LIN {X 0,Y 229.325,Z 211.915,A -85,B 0,C 180,E1 -20369.246,E2 -20369.246} C_VEL
LIN {X 0,Y 228.577,Z 208.445,A -85,B 0,C 180,E1 -20369.539,E2 -20369.539} C_VEL
LIN {X 0,Y 226.457,Z 198.769,A -85,B 0,C 180,E1 -20372.733,E2 -20372.733} C_VEL
LIN {X 0,Y 227.361,Z 200.21,A -85,B 0,C 180,E1 -20373.176,E2 -20373.176} C_VEL
LIN {X 0,Y 228.456,Z 200.617,A -85,B 0,C 180,E1 -20373.624,E2 -20373.624} C_VEL
LIN {X 0,Y 231.599,Z 199.766,A -85,B 0,C 180,E1 -20374.751,E2 -20374.751} C_VEL
LIN {X 0,Y 238.539,Z 200.37,A -85,B 0,C 180,E1 -20377.156,E2 -20377.156} C_VEL
LIN {X 0,Y 245.648,Z 210.634,A -85,B 0,C 180,E1 -20379.796,E2 -20379.796} C_VEL
LIN {X 0,Y 252.602,Z 221.645,A -85,B 0,C 180,E1 -20382.149,E2 -20382.149} C_VEL
LIN {X 0,Y 259.12,Z 233.125,A -85,B 0,C 180,E1 -20384.198,E2 -20384.198} C_VEL
LIN {X 0,Y 265.214,Z 245.318,A -85,B 0,C 180,E1 -20386.014,E2 -20386.014} C_VEL
LIN {X 0,Y 262.986,Z 287.428,A -85,B 0,C 180,E1 -20387.109,E2 -20387.109} C_VEL
LIN {X 0,Y 259.421,Z 351.334,A -85,B 0,C 180,E1 -20388.801,E2 -20388.801} C_VEL
LIN {X 0,Y 257.911,Z 366.77,A -85,B 0,C 180,E1 -20389.505,E2 -20389.505} C_VEL
LIN {X 0,Y 255.99,Z 381.125,A -85,B 0,C 180,E1 -20390.471,E2 -20390.471} C_VEL
LIN {X 0,Y 253.585,Z 394.744,A -85,B 0,C 180,E1 -20391.673,E2 -20391.673} C_VEL
LIN {X 0,Y 250.903,Z 406.648,A -85,B 0,C 180,E1 -20392.968,E2 -20392.968} C_VEL
LIN {X 0,Y 247.588,Z 419.265,A -85,B 0,C 180,E1 -20394.663,E2 -20394.663} C_VEL
LIN {X 0,Y 243.898,Z 430.94,A -85,B 0,C 180,E1 -20396.556,E2 -20396.556} C_VEL
LIN {X 0,Y 240.301,Z 441.724,A -85,B 0,C 180,E1 -20398.724,E2 -20398.724} C_VEL
LIN {X 0,Y 236.767,Z 451.626,A -85,B 0,C 180,E1 -20401.159,E2 -20401.159} C_VEL
LIN {X 0,Y 232.861,Z 461.299,A -85,B 0,C 180,E1 -20404.045,E2 -20404.045} C_VEL
LIN {X 0,Y 229.659,Z 468.909,A -85,B 0,C 180,E1 -20406.858,E2 -20406.858} C_VEL
LIN {X 0,Y 227.5,Z 474.158,A -85,B 0,C 180,E1 -20409.188,E2 -20409.188} C_VEL
LIN {X 0,Y 224.703,Z 480.638,A -85,B 0,C 180,E1 -20412.713,E2 -20412.713} C_VEL
LIN {X 0,Y 222.612,Z 485.689,A -85,B 0,C 180,E1 -20416.301,E2 -20416.301} C_VEL
LIN {X 0,Y 220.943,Z 489.84,A -85,B 0,C 180,E1 -20420.43,E2 -20420.43} C_VEL
LIN {X 0,Y 220.007,Z 492.412,A -85,B 0,C 180,E1 -20424.498,E2 -20424.498} C_VEL
LIN {X 0,Y 219.688,Z 493.551,A -85,B 0,C 180,E1 -20428.164,E2 -20428.164} C_VEL
LIN {X 0,Y 219.687,Z 493.562,A -85,B 0,C 180,E1 -20431.831,E2 -20431.831} C_VEL
LIN {X 0,Y 219.992,Z 492.468,A -85,B 0,C 180,E1 -20435.497,E2 -20435.497} C_VEL
LIN {X 0,Y 220.941,Z 489.942,A -85,B 0,C 180,E1 -20439.565,E2 -20439.565} C_VEL
LIN {X 0,Y 222.572,Z 485.851,A -85,B 0,C 180,E1 -20443.697,E2 -20443.697} C_VEL
LIN {X 0,Y 224.648,Z 480.852,A -85,B 0,C 180,E1 -20447.287,E2 -20447.287} C_VEL
LIN {X 0,Y 227.427,Z 474.422,A -85,B 0,C 180,E1 -20450.814,E2 -20450.814} C_VEL
LIN {X 0,Y 230.677,Z 466.604,A -85,B 0,C 180,E1 -20454.188,E2 -20454.188} C_VEL
LIN {X 0,Y 234.374,Z 457.762,A -85,B 0,C 180,E1 -20457.21,E2 -20457.21} C_VEL
LIN {X 0,Y 237.858,Z 448.945,A -85,B 0,C 180,E1 -20459.661,E2 -20459.661} C_VEL
LIN {X 0,Y 241.567,Z 438.263,A -85,B 0,C 180,E1 -20462.143,E2 -20462.143} C_VEL
LIN {X 0,Y 245.601,Z 426.051,A -85,B 0,C 180,E1 -20464.41,E2 -20464.41} C_VEL
LIN {X 0,Y 249.28,Z 413.399,A -85,B 0,C 180,E1 -20466.3,E2 -20466.3} C_VEL
LIN {X 0,Y 252.318,Z 401.135,A -85,B 0,C 180,E1 -20467.788,E2 -20467.788} C_VEL
LIN {X 0,Y 255.179,Z 386.887,A -85,B 0,C 180,E1 -20469.175,E2 -20469.175} C_VEL
LIN {X 0,Y 257.389,Z 371.923,A -85,B 0,C 180,E1 -20470.307,E2 -20470.307} C_VEL
LIN {X 0,Y 259.139,Z 356.374,A -85,B 0,C 180,E1 -20471.12,E2 -20471.12} C_VEL
LIN {X 0,Y 260.266,Z 339.563,A -85,B 0,C 180,E1 -20471.675,E2 -20471.675} C_VEL
LIN {X 0,Y 265.417,Z 246.396,A -85,B 0,C 180,E1 -20474.051,E2 -20474.051} C_VEL
LIN {X 0,Y 265.269,Z 245.25,A -85,B 0,C 180,E1 -20474.125,E2 -20474.125} C_VEL
LIN {X 0,Y 259.088,Z 232.99,A -85,B 0,C 180,E1 -20475.97,E2 -20475.97} C_VEL
LIN {X 0,Y 253.13,Z 222.402,A -85,B 0,C 180,E1 -20477.847,E2 -20477.847} C_VEL
LIN {X 0,Y 245.979,Z 211.094,A -85,B 0,C 180,E1 -20480.261,E2 -20480.261} C_VEL
LIN {X 0,Y 239.067,Z 201.088,A -85,B 0,C 180,E1 -20482.821,E2 -20482.821} C_VEL
LIN {X 0,Y 232.707,Z 192.573,A -85,B 0,C 180,E1 -20485.431,E2 -20485.431} C_VEL
LIN {X 0,Y 228.728,Z 187.686,A -85,B 0,C 180,E1 -20487.21,E2 -20487.21} C_VEL
LIN {X 0,Y 226.735,Z 185.16,A -85,B 0,C 180,E1 -20488.201,E2 -20488.201} C_VEL
LIN {X 0,Y 223.951,Z 180.168,A -85,B 0,C 180,E1 -20490.894,E2 -20490.894} C_VEL
LIN {X 0,Y 221.995,Z 177.687,A -85,B 0,C 180,E1 -20492.625,E2 -20492.625} C_VEL
LIN {X 0,Y 220.878,Z 174.575,A -85,B 0,C 180,E1 -20494.308,E2 -20494.308} C_VEL
LIN {X 0,Y 220.869,Z 174.594,A -85,B 0,C 180,E1 -20497.552,E2 -20497.552} C_VEL
LIN {X 0,Y 220.975,Z 174.567,A -85,B 0,C 180,E1 -20502.57,E2 -20502.57} C_VEL
LIN {X 0,Y 220.966,Z 174.571,A -85,B 0,C 180,E1 -20504.317,E2 -20504.317} C_VEL
LIN {X 0,Y 220.355,Z 174.642,A -85,B 0,C 180,E1 -20505.84,E2 -20505.84} C_VEL
LIN {X 0,Y 217.73,Z 174.971,A -85,B 0,C 180,E1 -20508.335,E2 -20508.335} C_VEL
LIN {X 0,Y 214.62,Z 175.364,A -85,B 0,C 180,E1 -20511.411,E2 -20511.411} C_VEL
LIN {X 0,Y 214.224,Z 175.396,A -85,B 0,C 180,E1 -20512.473,E2 -20512.473} C_VEL
LIN {X 0,Y 214.437,Z 175.381,A -85,B 0,C 180,E1 -20518.122,E2 -20518.122} C_VEL
LIN {X 0,Y 214.545,Z 175.35,A -85,B 0,C 180,E1 -20520,E2 -20520} C_VEL
LIN {X 0,Y 214.437,Z 175.375,A -85,B 0,C 180,E1 -20521.878,E2 -20521.878} C_VEL
LIN {X 0,Y 214.218,Z 175.391,A -85,B 0,C 180,E1 -20527.541,E2 -20527.541} C_VEL
LIN {X 0,Y 214.013,Z 175.427,A -85,B 0,C 180,E1 -20531.363,E2 -20531.363} C_VEL
LIN {X 0,Y 213.924,Z 175.445,A -85,B 0,C 180,E1 -20535.237,E2 -20535.237} C_VEL
LIN {X 0,Y 213.848,Z 175.441,A -85,B 0,C 180,E1 -20539.561,E2 -20539.561} C_VEL
LIN {X 0,Y 214.813,Z 178.313,A -85,B 0,C 180,E1 -20541.093,E2 -20541.093} C_VEL
LIN {X 0,Y 216.83,Z 180.388,A -85,B 0,C 180,E1 -20542.889,E2 -20542.889} C_VEL
LIN {X 0,Y 217.83,Z 181.739,A -85,B 0,C 180,E1 -20543.784,E2 -20543.784} C_VEL
LIN {X 0,Y 218.737,Z 183.542,A -85,B 0,C 180,E1 -20544.689,E2 -20544.689} C_VEL
LIN {X 0,Y 221.04,Z 186.119,A -85,B 0,C 180,E1 -20546.432,E2 -20546.432} C_VEL
LIN {X 0,Y 222.127,Z 188.36,A -85,B 0,C 180,E1 -20547.41,E2 -20547.41} C_VEL
LIN {X 0,Y 224.452,Z 191.343,A -85,B 0,C 180,E1 -20549.034,E2 -20549.034} C_VEL
LIN {X 0,Y 225.598,Z 193.42,A -85,B 0,C 180,E1 -20549.897,E2 -20549.897} C_VEL
LIN {X 0,Y 227.569,Z 196.049,A -85,B 0,C 180,E1 -20551.15,E2 -20551.15} C_VEL
LIN {X 0,Y 233.444,Z 205.295,A -85,B 0,C 180,E1 -20554.628,E2 -20554.628} C_VEL
LIN {X 0,Y 241.251,Z 216.448,A -85,B 0,C 180,E1 -20557.717,E2 -20557.717} C_VEL
LIN {X 0,Y 247.875,Z 232.788,A -85,B 0,C 180,E1 -20560.339,E2 -20560.339} C_VEL
LIN {X 0,Y 255.318,Z 252.374,A -85,B 0,C 180,E1 -20563.028,E2 -20563.028} C_VEL
LIN {X 0,Y 257.507,Z 289.946,A -85,B 0,C 180,E1 -20564.995,E2 -20564.995} C_VEL
LIN {X 0,Y 252.092,Z 383.718,A -85,B 0,C 180,E1 -20567.467,E2 -20567.467} C_VEL
LIN {X 0,Y 250.136,Z 399.638,A -85,B 0,C 180,E1 -20568.144,E2 -20568.144} C_VEL
LIN {X 0,Y 247.405,Z 414.728,A -85,B 0,C 180,E1 -20569.074,E2 -20569.074} C_VEL
LIN {X 0,Y 244.31,Z 428.33,A -85,B 0,C 180,E1 -20570.207,E2 -20570.207} C_VEL
LIN {X 0,Y 240.594,Z 441.726,A -85,B 0,C 180,E1 -20571.633,E2 -20571.633} C_VEL
LIN {X 0,Y 236.89,Z 453.76,A -85,B 0,C 180,E1 -20573.268,E2 -20573.268} C_VEL
LIN {X 0,Y 232.819,Z 465.673,A -85,B 0,C 180,E1 -20575.269,E2 -20575.269} C_VEL
LIN {X 0,Y 228.753,Z 476.424,A -85,B 0,C 180,E1 -20577.479,E2 -20577.479} C_VEL
LIN {X 0,Y 224.933,Z 486.407,A -85,B 0,C 180,E1 -20580.008,E2 -20580.008} C_VEL
LIN {X 0,Y 221.038,Z 496.178,A -85,B 0,C 180,E1 -20583.057,E2 -20583.057} C_VEL
LIN {X 0,Y 217.946,Z 504.37,A -85,B 0,C 180,E1 -20586.232,E2 -20586.232} C_VEL
LIN {X 0,Y 215.071,Z 512.016,A -85,B 0,C 180,E1 -20589.936,E2 -20589.936} C_VEL
LIN {X 0,Y 213.19,Z 518.129,A -85,B 0,C 180,E1 -20593.73,E2 -20593.73} C_VEL
LIN {X 0,Y 212.09,Z 522.843,A -85,B 0,C 180,E1 -20597.564,E2 -20597.564} C_VEL
LIN {X 0,Y 211.82,Z 525.486,A -85,B 0,C 180,E1 -20600.453,E2 -20600.453} C_VEL
LIN {X 0,Y 212.066,Z 527.982,A -85,B 0,C 180,E1 -20604.297,E2 -20604.297} C_VEL
LIN {X 0,Y 212.353,Z 529.246,A -85,B 0,C 180,E1 -20608.106,E2 -20608.106} C_VEL
LIN {X 0,Y 212.626,Z 529.429,A -85,B 0,C 180,E1 -20610.002,E2 -20610.002} C_VEL
LIN {X 0,Y 212.167,Z 528.752,A -85,B 0,C 180,E1 -20613.801,E2 -20613.801} C_VEL
LIN {X 0,Y 212.076,Z 527.748,A -85,B 0,C 180,E1 -20616.19,E2 -20616.19} C_VEL
LIN {X 0,Y 211.873,Z 525.455,A -85,B 0,C 180,E1 -20619.549,E2 -20619.549} C_VEL
LIN {X 0,Y 212.333,Z 521.705,A -85,B 0,C 180,E1 -20623.399,E2 -20623.399} C_VEL
LIN {X 0,Y 213.71,Z 516.214,A -85,B 0,C 180,E1 -20627.507,E2 -20627.507} C_VEL
LIN {X 0,Y 215.718,Z 510.154,A -85,B 0,C 180,E1 -20631.003,E2 -20631.003} C_VEL
LIN {X 0,Y 218.799,Z 502.051,A -85,B 0,C 180,E1 -20634.684,E2 -20634.684} C_VEL
LIN {X 0,Y 221.957,Z 493.814,A -85,B 0,C 180,E1 -20637.721,E2 -20637.721} C_VEL
LIN {X 0,Y 226.494,Z 488.538,A -85,B 0,C 180,E1 -20640.799,E2 -20640.799} C_VEL
LIN {X 0,Y 234.217,Z 479.658,A -85,B 0,C 180,E1 -20644.761,E2 -20644.761} C_VEL
LIN {X 0,Y 239.708,Z 473.405,A -85,B 0,C 180,E1 -20646.947,E2 -20646.947} C_VEL
LIN {X 0,Y 247.844,Z 463.784,A -85,B 0,C 180,E1 -20649.647,E2 -20649.647} C_VEL
LIN {X 0,Y 255.71,Z 454.035,A -85,B 0,C 180,E1 -20651.799,E2 -20651.799} C_VEL
LIN {X 0,Y 264.235,Z 442.772,A -85,B 0,C 180,E1 -20653.754,E2 -20653.754} C_VEL
LIN {X 0,Y 272.732,Z 430.571,A -85,B 0,C 180,E1 -20655.389,E2 -20655.389} C_VEL
LIN {X 0,Y 281.83,Z 416.056,A -85,B 0,C 180,E1 -20656.839,E2 -20656.839} C_VEL
LIN {X 0,Y 289.18,Z 402.986,A -85,B 0,C 180,E1 -20657.84,E2 -20657.84} C_VEL
LIN {X 0,Y 295.883,Z 389.316,A -85,B 0,C 180,E1 -20658.653,E2 -20658.653} C_VEL
LIN {X 0,Y 296.103,Z 388.689,A -85,B 0,C 180,E1 -20658.973,E2 -20658.973} C_VEL
LIN {X 0,Y 288.903,Z 401.868,A -85,B 0,C 180,E1 -20660.315,E2 -20660.315} C_VEL
LIN {X 0,Y 282.68,Z 411.802,A -85,B 0,C 180,E1 -20661.571,E2 -20661.571} C_VEL
LIN {X 0,Y 274.659,Z 423.047,A -85,B 0,C 180,E1 -20663.383,E2 -20663.383} C_VEL
LIN {X 0,Y 265.94,Z 433.664,A -85,B 0,C 180,E1 -20665.606,E2 -20665.606} C_VEL
LIN {X 0,Y 258.302,Z 441.797,A -85,B 0,C 180,E1 -20667.842,E2 -20667.842} C_VEL
LIN {X 0,Y 250.363,Z 449.136,A -85,B 0,C 180,E1 -20670.578,E2 -20670.578} C_VEL
LIN {X 0,Y 243.225,Z 454.724,A -85,B 0,C 180,E1 -20673.393,E2 -20673.393} C_VEL
LIN {X 0,Y 238.278,Z 457.888,A -85,B 0,C 180,E1 -20675.611,E2 -20675.611} C_VEL
LIN {X 0,Y 232.447,Z 460.848,A -85,B 0,C 180,E1 -20678.727,E2 -20678.727} C_VEL
LIN {X 0,Y 227.254,Z 462.372,A -85,B 0,C 180,E1 -20681.986,E2 -20681.986} C_VEL
LIN {X 0,Y 222.965,Z 462.441,A -85,B 0,C 180,E1 -20685.395,E2 -20685.395} C_VEL
LIN {X 0,Y 221.026,Z 461.966,A -85,B 0,C 180,E1 -20687.14,E2 -20687.14} C_VEL
LIN {X 0,Y 218.058,Z 459.857,A -85,B 0,C 180,E1 -20690.727,E2 -20690.727} C_VEL
LIN {X 0,Y 217.006,Z 458.242,A -85,B 0,C 180,E1 -20692.557,E2 -20692.557} C_VEL
LIN {X 0,Y 215.507,Z 455.078,A -85,B 0,C 180,E1 -20695.324,E2 -20695.324} C_VEL
LIN {X 0,Y 214.393,Z 451,A -85,B 0,C 180,E1 -20698.122,E2 -20698.122} C_VEL
LIN {X 0,Y 213.83,Z 445.923,A -85,B 0,C 180,E1 -20700.942,E2 -20700.942} C_VEL
LIN {X 0,Y 213.595,Z 438.597,A -85,B 0,C 180,E1 -20704.246,E2 -20704.246} C_VEL
LIN {X 0,Y 213.747,Z 430.934,A -85,B 0,C 180,E1 -20707.083,E2 -20707.083} C_VEL
LIN {X 0,Y 214.115,Z 422.636,A -85,B 0,C 180,E1 -20709.659,E2 -20709.659} C_VEL
LIN {X 0,Y 214.927,Z 411.615,A -85,B 0,C 180,E1 -20712.512,E2 -20712.512} C_VEL
LIN {X 0,Y 215.878,Z 399.483,A -85,B 0,C 180,E1 -20715.097,E2 -20715.097} C_VEL
LIN {X 0,Y 216.932,Z 385.995,A -85,B 0,C 180,E1 -20717.438,E2 -20717.438} C_VEL
LIN {X 0,Y 217.982,Z 372.874,A -85,B 0,C 180,E1 -20719.298,E2 -20719.298} C_VEL
LIN {X 0,Y 218.938,Z 358.222,A -85,B 0,C 180,E1 -20720.95,E2 -20720.95} C_VEL
LIN {X 0,Y 219.873,Z 342.126,A -85,B 0,C 180,E1 -20722.334,E2 -20722.334} C_VEL
LIN {X 0,Y 220.648,Z 323.641,A -85,B 0,C 180,E1 -20723.463,E2 -20723.463} C_VEL
LIN {X 0,Y 225.363,Z 240.466,A -85,B 0,C 180,E1 -20727.931,E2 -20727.931} C_VEL
LIN {X 0,Y 222.713,Z 215.537,A -85,B 0,C 180,E1 -20729.508,E2 -20729.508} C_VEL
LIN {X 0,Y 222.134,Z 211.353,A -85,B 0,C 180,E1 -20729.784,E2 -20729.784} C_VEL
LIN {X 0,Y 221.452,Z 208.945,A -85,B 0,C 180,E1 -20729.978,E2 -20729.978} C_VEL
LIN {X 0,Y 220.886,Z 206.421,A -85,B 0,C 180,E1 -20730.851,E2 -20730.851} C_VEL
LIN {X 0,Y 221.713,Z 207.774,A -85,B 0,C 180,E1 -20731.298,E2 -20731.298} C_VEL
LIN {X 0,Y 224.409,Z 207.769,A -85,B 0,C 180,E1 -20732.432,E2 -20732.432} C_VEL
LIN {X 0,Y 225.53,Z 207.062,A -85,B 0,C 180,E1 -20732.845,E2 -20732.845} C_VEL
LIN {X 0,Y 227.735,Z 207.662,A -85,B 0,C 180,E1 -20733.745,E2 -20733.745} C_VEL
LIN {X 0,Y 230.723,Z 206.919,A -85,B 0,C 180,E1 -20734.819,E2 -20734.819} C_VEL
LIN {X 0,Y 236.416,Z 207.35,A -85,B 0,C 180,E1 -20736.812,E2 -20736.812} C_VEL
LIN {X 0,Y 244.041,Z 218.717,A -85,B 0,C 180,E1 -20739.703,E2 -20739.703} C_VEL
LIN {X 0,Y 250.616,Z 229.722,A -85,B 0,C 180,E1 -20741.98,E2 -20741.98} C_VEL
LIN {X 0,Y 256.73,Z 241.001,A -85,B 0,C 180,E1 -20743.952,E2 -20743.952} C_VEL
LIN {X 0,Y 260.117,Z 247.984,A -85,B 0,C 180,E1 -20745.004,E2 -20745.004} C_VEL
LIN {X 0,Y 254.259,Z 350.477,A -85,B 0,C 180,E1 -20747.707,E2 -20747.707} C_VEL
LIN {X 0,Y 252.721,Z 366.071,A -85,B 0,C 180,E1 -20748.396,E2 -20748.396} C_VEL
LIN {X 0,Y 250.968,Z 379.134,A -85,B 0,C 180,E1 -20749.248,E2 -20749.248} C_VEL
LIN {X 0,Y 248.48,Z 393.395,A -85,B 0,C 180,E1 -20750.475,E2 -20750.475} C_VEL
LIN {X 0,Y 245.301,Z 407.222,A -85,B 0,C 180,E1 -20751.974,E2 -20751.974} C_VEL
LIN {X 0,Y 241.862,Z 419.842,A -85,B 0,C 180,E1 -20753.695,E2 -20753.695} C_VEL
LIN {X 0,Y 238.025,Z 431.519,A -85,B 0,C 180,E1 -20755.617,E2 -20755.617} C_VEL
LIN {X 0,Y 234.28,Z 442.306,A -85,B 0,C 180,E1 -20757.825,E2 -20757.825} C_VEL
LIN {X 0,Y 230.603,Z 452.208,A -85,B 0,C 180,E1 -20760.312,E2 -20760.312} C_VEL
LIN {X 0,Y 226.517,Z 461.883,A -85,B 0,C 180,E1 -20763.262,E2 -20763.262} C_VEL
LIN {X 0,Y 223.027,Z 469.78,A -85,B 0,C 180,E1 -20766.258,E2 -20766.258} C_VEL
LIN {X 0,Y 220.896,Z 474.743,A -85,B 0,C 180,E1 -20768.536,E2 -20768.536} C_VEL
LIN {X 0,Y 217.947,Z 481.223,A -85,B 0,C 180,E1 -20772.159,E2 -20772.159} C_VEL
LIN {X 0,Y 215.744,Z 486.274,A -85,B 0,C 180,E1 -20775.856,E2 -20775.856} C_VEL
LIN {X 0,Y 213.942,Z 490.51,A -85,B 0,C 180,E1 -20780.233,E2 -20780.233} C_VEL
LIN {X 0,Y 212.954,Z 492.998,A -85,B 0,C 180,E1 -20784.316,E2 -20784.316} C_VEL
LIN {X 0,Y 212.625,Z 494.136,A -85,B 0,C 180,E1 -20788.103,E2 -20788.103} C_VEL
LIN {X 0,Y 212.624,Z 494.146,A -85,B 0,C 180,E1 -20791.892,E2 -20791.892} C_VEL
LIN {X 0,Y 212.938,Z 493.053,A -85,B 0,C 180,E1 -20795.68,E2 -20795.68} C_VEL
LIN {X 0,Y 213.939,Z 490.612,A -85,B 0,C 180,E1 -20799.762,E2 -20799.762} C_VEL
LIN {X 0,Y 215.707,Z 486.434,A -85,B 0,C 180,E1 -20804.141,E2 -20804.141} C_VEL
LIN {X 0,Y 217.896,Z 481.435,A -85,B 0,C 180,E1 -20807.84,E2 -20807.84} C_VEL
LIN {X 0,Y 220.813,Z 475.005,A -85,B 0,C 180,E1 -20811.468,E2 -20811.468} C_VEL
LIN {X 0,Y 223.842,Z 468.05,A -85,B 0,C 180,E1 -20814.58,E2 -20814.58} C_VEL
LIN {X 0,Y 227.54,Z 459.654,A -85,B 0,C 180,E1 -20817.598,E2 -20817.598} C_VEL
LIN {X 0,Y 231.727,Z 449.523,A -85,B 0,C 180,E1 -20820.528,E2 -20820.528} C_VEL
LIN {X 0,Y 235.499,Z 439.099,A -85,B 0,C 180,E1 -20823.005,E2 -20823.005} C_VEL
LIN {X 0,Y 239.42,Z 427.764,A -85,B 0,C 180,E1 -20825.172,E2 -20825.172} C_VEL
LIN {X 0,Y 243.216,Z 415.352,A -85,B 0,C 180,E1 -20827.097,E2 -20827.097} C_VEL
LIN {X 0,Y 246.783,Z 401.695,A -85,B 0,C 180,E1 -20828.791,E2 -20828.791} C_VEL
LIN {X 0,Y 249.741,Z 387.44,A -85,B 0,C 180,E1 -20830.199,E2 -20830.199} C_VEL
LIN {X 0,Y 252.028,Z 372.654,A -85,B 0,C 180,E1 -20831.331,E2 -20831.331} C_VEL
LIN {X 0,Y 253.75,Z 357.955,A -85,B 0,C 180,E1 -20832.124,E2 -20832.124} C_VEL
LIN {X 0,Y 254.924,Z 341.798,A -85,B 0,C 180,E1 -20832.686,E2 -20832.686} C_VEL
LIN {X 0,Y 260.239,Z 249.198,A -85,B 0,C 180,E1 -20835.074,E2 -20835.074} C_VEL
LIN {X 0,Y 260.088,Z 247.786,A -85,B 0,C 180,E1 -20835.163,E2 -20835.163} C_VEL
LIN {X 0,Y 252.607,Z 233.061,A -85,B 0,C 180,E1 -20837.534,E2 -20837.534} C_VEL
LIN {X 0,Y 245.102,Z 220.399,A -85,B 0,C 180,E1 -20840.089,E2 -20840.089} C_VEL
LIN {X 0,Y 237.859,Z 209.323,A -85,B 0,C 180,E1 -20842.803,E2 -20842.803} C_VEL
LIN {X 0,Y 230.351,Z 198.968,A -85,B 0,C 180,E1 -20845.95,E2 -20845.95} C_VEL
LIN {X 0,Y 226.333,Z 193.932,A -85,B 0,C 180,E1 -20847.81,E2 -20847.81} C_VEL
LIN {X 0,Y 220.058,Z 186.147,A -85,B 0,C 180,E1 -20851.115,E2 -20851.115} C_VEL
LIN {X 0,Y 216.45,Z 180.115,A -85,B 0,C 180,E1 -20855.032,E2 -20855.032} C_VEL
LIN {X 0,Y 214.688,Z 178.092,A -85,B 0,C 180,E1 -20856.869,E2 -20856.869} C_VEL
LIN {X 0,Y 213.816,Z 175.471,A -85,B 0,C 180,E1 -20858.551,E2 -20858.551} C_VEL
LIN {X 0,Y 213.934,Z 175.446,A -85,B 0,C 180,E1 -20862.803,E2 -20862.803} C_VEL
LIN {X 0,Y 213.944,Z 175.429,A -85,B 0,C 180,E1 -20866.706,E2 -20866.706} C_VEL
LIN {X 0,Y 214.187,Z 175.43,A -85,B 0,C 180,E1 -20870.557,E2 -20870.557} C_VEL
LIN {X 0,Y 214.224,Z 175.396,A -85,B 0,C 180,E1 -20872.473,E2 -20872.473} C_VEL
LIN {X 0,Y 213.476,Z 175.494,A -85,B 0,C 180,E1 -20874.043,E2 -20874.043} C_VEL
LIN {X 0,Y 210.782,Z 175.854,A -85,B 0,C 180,E1 -20876.616,E2 -20876.616} C_VEL
LIN {X 0,Y 207.763,Z 176.198,A -85,B 0,C 180,E1 -20879.793,E2 -20879.793} C_VEL
LIN {X 0,Y 207.418,Z 176.239,A -85,B 0,C 180,E1 -20880.888,E2 -20880.888} C_VEL
LIN {X 0,Y 207.158,Z 176.272,A -85,B 0,C 180,E1 -20887.799,E2 -20887.799} C_VEL
LIN {X 0,Y 206.933,Z 176.303,A -85,B 0,C 180,E1 -20891.758,E2 -20891.758} C_VEL
LIN {X 0,Y 206.867,Z 176.309,A -85,B 0,C 180,E1 -20893.883,E2 -20893.883} C_VEL
LIN {X 0,Y 207.707,Z 178.867,A -85,B 0,C 180,E1 -20895.705,E2 -20895.705} C_VEL
LIN {X 0,Y 210.87,Z 182.464,A -85,B 0,C 180,E1 -20899.468,E2 -20899.468} C_VEL
LIN {X 0,Y 212.403,Z 185.386,A -85,B 0,C 180,E1 -20901.344,E2 -20901.344} C_VEL
LIN {X 0,Y 214.427,Z 187.58,A -85,B 0,C 180,E1 -20903.16,E2 -20903.16} C_VEL
LIN {X 0,Y 216.38,Z 190.752,A -85,B 0,C 180,E1 -20904.976,E2 -20904.976} C_VEL
LIN {X 0,Y 217.543,Z 192.015,A -85,B 0,C 180,E1 -20905.857,E2 -20905.857} C_VEL
LIN {X 0,Y 221.452,Z 198.204,A -85,B 0,C 180,E1 -20908.945,E2 -20908.945} C_VEL
LIN {X 0,Y 224.855,Z 203.404,A -85,B 0,C 180,E1 -20911.264,E2 -20911.264} C_VEL
LIN {X 0,Y 231.578,Z 212.565,A -85,B 0,C 180,E1 -20914.353,E2 -20914.353} C_VEL
LIN {X 0,Y 237.84,Z 221.883,A -85,B 0,C 180,E1 -20916.924,E2 -20916.924} C_VEL
LIN {X 0,Y 243.842,Z 237.132,A -85,B 0,C 180,E1 -20919.424,E2 -20919.424} C_VEL
LIN {X 0,Y 250.561,Z 255.319,A -85,B 0,C 180,E1 -20921.991,E2 -20921.991} C_VEL
LIN {X 0,Y 252.46,Z 290.921,A -85,B 0,C 180,E1 -20923.895,E2 -20923.895} C_VEL
LIN {X 0,Y 246.906,Z 383.227,A -85,B 0,C 180,E1 -20926.353,E2 -20926.353} C_VEL
LIN {X 0,Y 244.885,Z 399.101,A -85,B 0,C 180,E1 -20927.034,E2 -20927.034} C_VEL
LIN {X 0,Y 242.069,Z 414.173,A -85,B 0,C 180,E1 -20927.969,E2 -20927.969} C_VEL
LIN {X 0,Y 238.886,Z 427.768,A -85,B 0,C 180,E1 -20929.115,E2 -20929.115} C_VEL
LIN {X 0,Y 235.062,Z 441.158,A -85,B 0,C 180,E1 -20930.558,E2 -20930.558} C_VEL
LIN {X 0,Y 231.052,Z 453.579,A -85,B 0,C 180,E1 -20932.265,E2 -20932.265} C_VEL
LIN {X 0,Y 226.576,Z 466.164,A -85,B 0,C 180,E1 -20934.441,E2 -20934.441} C_VEL
LIN {X 0,Y 222.046,Z 477.635,A -85,B 0,C 180,E1 -20936.911,E2 -20936.911} C_VEL
LIN {X 0,Y 218.118,Z 487.322,A -85,B 0,C 180,E1 -20939.507,E2 -20939.507} C_VEL
LIN {X 0,Y 214.13,Z 496.849,A -85,B 0,C 180,E1 -20942.648,E2 -20942.648} C_VEL
LIN {X 0,Y 210.938,Z 504.806,A -85,B 0,C 180,E1 -20945.915,E2 -20945.915} C_VEL
LIN {X 0,Y 208.313,Z 511.423,A -85,B 0,C 180,E1 -20949.256,E2 -20949.256} C_VEL
LIN {X 0,Y 206.288,Z 517.535,A -85,B 0,C 180,E1 -20953.17,E2 -20953.17} C_VEL
LIN {X 0,Y 205.094,Z 522.251,A -85,B 0,C 180,E1 -20957.133,E2 -20957.133} C_VEL
LIN {X 0,Y 204.755,Z 524.894,A -85,B 0,C 180,E1 -20960.121,E2 -20960.121} C_VEL
LIN {X 0,Y 204.986,Z 527.394,A -85,B 0,C 180,E1 -20964.099,E2 -20964.099} C_VEL
LIN {X 0,Y 205.257,Z 528.659,A -85,B 0,C 180,E1 -20968.04,E2 -20968.04} C_VEL
LIN {X 0,Y 205.566,Z 528.846,A -85,B 0,C 180,E1 -20970.002,E2 -20970.002} C_VEL
LIN {X 0,Y 205.092,Z 528.166,A -85,B 0,C 180,E1 -20973.932,E2 -20973.932} C_VEL
LIN {X 0,Y 205.002,Z 527.259,A -85,B 0,C 180,E1 -20976.178,E2 -20976.178} C_VEL
LIN {X 0,Y 204.801,Z 524.862,A -85,B 0,C 180,E1 -20979.882,E2 -20979.882} C_VEL
LIN {X 0,Y 205.325,Z 521.109,A -85,B 0,C 180,E1 -20983.865,E2 -20983.865} C_VEL
LIN {X 0,Y 206.702,Z 516.048,A -85,B 0,C 180,E1 -20987.821,E2 -20987.821} C_VEL
LIN {X 0,Y 208.992,Z 509.558,A -85,B 0,C 180,E1 -20991.712,E2 -20991.712} C_VEL
LIN {X 0,Y 212.236,Z 501.453,A -85,B 0,C 180,E1 -20995.501,E2 -20995.501} C_VEL
LIN {X 0,Y 215.308,Z 494.024,A -85,B 0,C 180,E1 -20998.369,E2 -20998.369} C_VEL
LIN {X 0,Y 221.917,Z 487.211,A -85,B 0,C 180,E1 -21002.576,E2 -21002.576} C_VEL
LIN {X 0,Y 230.264,Z 478.521,A -85,B 0,C 180,E1 -21006.527,E2 -21006.527} C_VEL
LIN {X 0,Y 237.218,Z 471.3,A -85,B 0,C 180,E1 -21009.021,E2 -21009.021} C_VEL
LIN {X 0,Y 245.898,Z 461.763,A -85,B 0,C 180,E1 -21011.647,E2 -21011.647} C_VEL
LIN {X 0,Y 255.499,Z 450.582,A -85,B 0,C 180,E1 -21013.994,E2 -21013.994} C_VEL
LIN {X 0,Y 264.619,Z 439.14,A -85,B 0,C 180,E1 -21015.817,E2 -21015.817} C_VEL
LIN {X 0,Y 273.695,Z 426.675,A -85,B 0,C 180,E1 -21017.313,E2 -21017.313} C_VEL
LIN {X 0,Y 282.456,Z 413.198,A -85,B 0,C 180,E1 -21018.555,E2 -21018.555} C_VEL
LIN {X 0,Y 286.281,Z 406.867,A -85,B 0,C 180,E1 -21019.018,E2 -21019.018} C_VEL
LIN {X 0,Y 285.92,Z 407.257,A -85,B 0,C 180,E1 -21019.355,E2 -21019.355} C_VEL
LIN {X 0,Y 278.202,Z 418.236,A -85,B 0,C 180,E1 -21020.835,E2 -21020.835} C_VEL
LIN {X 0,Y 269.619,Z 428.873,A -85,B 0,C 180,E1 -21022.696,E2 -21022.696} C_VEL
LIN {X 0,Y 261.472,Z 437.691,A -85,B 0,C 180,E1 -21024.698,E2 -21024.698} C_VEL
LIN {X 0,Y 254.865,Z 444.089,A -85,B 0,C 180,E1 -21026.53,E2 -21026.53} C_VEL
LIN {X 0,Y 246.716,Z 451.01,A -85,B 0,C 180,E1 -21029.153,E2 -21029.153} C_VEL
LIN {X 0,Y 239.163,Z 456.431,A -85,B 0,C 180,E1 -21031.955,E2 -21031.955} C_VEL
LIN {X 0,Y 232.208,Z 460.376,A -85,B 0,C 180,E1 -21034.93,E2 -21034.93} C_VEL
LIN {X 0,Y 226.114,Z 462.856,A -85,B 0,C 180,E1 -21038.101,E2 -21038.101} C_VEL
LIN {X 0,Y 220.699,Z 463.995,A -85,B 0,C 180,E1 -21041.431,E2 -21041.431} C_VEL
LIN {X 0,Y 216.236,Z 463.721,A -85,B 0,C 180,E1 -21044.929,E2 -21044.929} C_VEL
LIN {X 0,Y 214.215,Z 463.056,A -85,B 0,C 180,E1 -21046.723,E2 -21046.723} C_VEL
LIN {X 0,Y 211.114,Z 460.559,A -85,B 0,C 180,E1 -21050.419,E2 -21050.419} C_VEL
LIN {X 0,Y 209.404,Z 457.749,A -85,B 0,C 180,E1 -21053.254,E2 -21053.254} C_VEL
LIN {X 0,Y 207.69,Z 452.559,A -85,B 0,C 180,E1 -21057.091,E2 -21057.091} C_VEL
LIN {X 0,Y 206.794,Z 447.55,A -85,B 0,C 180,E1 -21060,E2 -21060} C_VEL
LIN {X 0,Y 206.524,Z 441.468,A -85,B 0,C 180,E1 -21062.926,E2 -21062.926} C_VEL
LIN {X 0,Y 206.468,Z 434.131,A -85,B 0,C 180,E1 -21065.861,E2 -21065.861} C_VEL
LIN {X 0,Y 206.973,Z 425.366,A -85,B 0,C 180,E1 -21068.79,E2 -21068.79} C_VEL
LIN {X 0,Y 207.602,Z 414.848,A -85,B 0,C 180,E1 -21071.72,E2 -21071.72} C_VEL
LIN {X 0,Y 208.454,Z 403.158,A -85,B 0,C 180,E1 -21074.398,E2 -21074.398} C_VEL
LIN {X 0,Y 209.474,Z 390.355,A -85,B 0,C 180,E1 -21076.821,E2 -21076.821} C_VEL
LIN {X 0,Y 210.525,Z 378.032,A -85,B 0,C 180,E1 -21078.743,E2 -21078.743} C_VEL
LIN {X 0,Y 211.517,Z 363.655,A -85,B 0,C 180,E1 -21080.546,E2 -21080.546} C_VEL
LIN {X 0,Y 212.476,Z 348.593,A -85,B 0,C 180,E1 -21082.027,E2 -21082.027} C_VEL
LIN {X 0,Y 213.226,Z 331.573,A -85,B 0,C 180,E1 -21083.252,E2 -21083.252} C_VEL
LIN {X 0,Y 217.869,Z 251.933,A -85,B 0,C 180,E1 -21087.727,E2 -21087.727} C_VEL
LIN {X 0,Y 218.34,Z 240.421,A -85,B 0,C 180,E1 -21088.37,E2 -21088.37} C_VEL
LIN {X 0,Y 216.267,Z 220.822,A -85,B 0,C 180,E1 -21089.669,E2 -21089.669} C_VEL
LIN {X 0,Y 217.029,Z 221.648,A -85,B 0,C 180,E1 -21090.082,E2 -21090.082} C_VEL
LIN {X 0,Y 218.11,Z 220.934,A -85,B 0,C 180,E1 -21090.532,E2 -21090.532} C_VEL
LIN {X 0,Y 219.709,Z 217.991,A -85,B 0,C 180,E1 -21091.06,E2 -21091.06} C_VEL
LIN {X 0,Y 220.91,Z 214.973,A -85,B 0,C 180,E1 -21091.396,E2 -21091.396} C_VEL
LIN {X 0,Y 224.153,Z 214.766,A -85,B 0,C 180,E1 -21092.742,E2 -21092.742} C_VEL
LIN {X 0,Y 225.138,Z 214.347,A -85,B 0,C 180,E1 -21093.113,E2 -21093.113} C_VEL
LIN {X 0,Y 227.997,Z 214.61,A -85,B 0,C 180,E1 -21094.233,E2 -21094.233} C_VEL
LIN {X 0,Y 231.027,Z 214.002,A -85,B 0,C 180,E1 -21095.31,E2 -21095.31} C_VEL
LIN {X 0,Y 234.185,Z 214.213,A -85,B 0,C 180,E1 -21096.416,E2 -21096.416} C_VEL
LIN {X 0,Y 240.868,Z 224.431,A -85,B 0,C 180,E1 -21099.038,E2 -21099.038} C_VEL
LIN {X 0,Y 247.876,Z 236.465,A -85,B 0,C 180,E1 -21101.552,E2 -21101.552} C_VEL
LIN {X 0,Y 254.87,Z 250.2,A -85,B 0,C 180,E1 -21103.881,E2 -21103.881} C_VEL
LIN {X 0,Y 255.038,Z 250.507,A -85,B 0,C 180,E1 -21103.933,E2 -21103.933} C_VEL
LIN {X 0,Y 249.071,Z 351.002,A -85,B 0,C 180,E1 -21106.612,E2 -21106.612} C_VEL
LIN {X 0,Y 247.48,Z 366.688,A -85,B 0,C 180,E1 -21107.315,E2 -21107.315} C_VEL
LIN {X 0,Y 245.372,Z 381.439,A -85,B 0,C 180,E1 -21108.304,E2 -21108.304} C_VEL
LIN {X 0,Y 242.662,Z 395.884,A -85,B 0,C 180,E1 -21109.605,E2 -21109.605} C_VEL
LIN {X 0,Y 239.328,Z 409.332,A -85,B 0,C 180,E1 -21111.118,E2 -21111.118} C_VEL
LIN {X 0,Y 235.798,Z 421.674,A -85,B 0,C 180,E1 -21112.873,E2 -21112.873} C_VEL
LIN {X 0,Y 231.849,Z 433.139,A -85,B 0,C 180,E1 -21114.832,E2 -21114.832} C_VEL
LIN {X 0,Y 227.68,Z 444.615,A -85,B 0,C 180,E1 -21117.301,E2 -21117.301} C_VEL
LIN {X 0,Y 223.837,Z 454.255,A -85,B 0,C 180,E1 -21119.841,E2 -21119.841} C_VEL
LIN {X 0,Y 219.649,Z 463.675,A -85,B 0,C 180,E1 -21122.872,E2 -21122.872} C_VEL
LIN {X 0,Y 216.424,Z 470.646,A -85,B 0,C 180,E1 -21125.619,E2 -21125.619} C_VEL
LIN {X 0,Y 213.395,Z 477.084,A -85,B 0,C 180,E1 -21128.758,E2 -21128.758} C_VEL
LIN {X 0,Y 210.568,Z 483.18,A -85,B 0,C 180,E1 -21132.517,E2 -21132.517} C_VEL
LIN {X 0,Y 208.383,Z 487.885,A -85,B 0,C 180,E1 -21136.342,E2 -21136.342} C_VEL
LIN {X 0,Y 206.861,Z 491.323,A -85,B 0,C 180,E1 -21140.217,E2 -21140.217} C_VEL
LIN {X 0,Y 205.904,Z 493.584,A -85,B 0,C 180,E1 -21144.12,E2 -21144.12} C_VEL
LIN {X 0,Y 205.564,Z 494.72,A -85,B 0,C 180,E1 -21148.038,E2 -21148.038} C_VEL
LIN {X 0,Y 205.562,Z 494.73,A -85,B 0,C 180,E1 -21151.957,E2 -21151.957} C_VEL
LIN {X 0,Y 205.888,Z 493.639,A -85,B 0,C 180,E1 -21155.875,E2 -21155.875} C_VEL
LIN {X 0,Y 206.94,Z 491.28,A -85,B 0,C 180,E1 -21159.974,E2 -21159.974} C_VEL
LIN {X 0,Y 208.834,Z 487.019,A -85,B 0,C 180,E1 -21164.617,E2 -21164.617} C_VEL
LIN {X 0,Y 211.147,Z 482.02,A -85,B 0,C 180,E1 -21168.431,E2 -21168.431} C_VEL
LIN {X 0,Y 214.231,Z 475.588,A -85,B 0,C 180,E1 -21172.162,E2 -21172.162} C_VEL
LIN {X 0,Y 217.411,Z 468.632,A -85,B 0,C 180,E1 -21175.358,E2 -21175.358} C_VEL
LIN {X 0,Y 221.288,Z 460.234,A -85,B 0,C 180,E1 -21178.447,E2 -21178.447} C_VEL
LIN {X 0,Y 225.651,Z 450.102,A -85,B 0,C 180,E1 -21181.442,E2 -21181.442} C_VEL
LIN {X 0,Y 229.536,Z 439.827,A -85,B 0,C 180,E1 -21183.935,E2 -21183.935} C_VEL
LIN {X 0,Y 233.67,Z 428.336,A -85,B 0,C 180,E1 -21186.172,E2 -21186.172} C_VEL
LIN {X 0,Y 237.623,Z 415.919,A -85,B 0,C 180,E1 -21188.124,E2 -21188.124} C_VEL
LIN {X 0,Y 241.324,Z 402.255,A -85,B 0,C 180,E1 -21189.841,E2 -21189.841} C_VEL
LIN {X 0,Y 244.382,Z 387.993,A -85,B 0,C 180,E1 -21191.269,E2 -21191.269} C_VEL
LIN {X 0,Y 246.754,Z 373.321,A -85,B 0,C 180,E1 -21192.405,E2 -21192.405} C_VEL
LIN {X 0,Y 248.56,Z 358.467,A -85,B 0,C 180,E1 -21193.215,E2 -21193.215} C_VEL
LIN {X 0,Y 249.78,Z 342.251,A -85,B 0,C 180,E1 -21193.784,E2 -21193.784} C_VEL
LIN {X 0,Y 255.179,Z 251.518,A -85,B 0,C 180,E1 -21196.15,E2 -21196.15} C_VEL
LIN {X 0,Y 254.871,Z 250.031,A -85,B 0,C 180,E1 -21196.283,E2 -21196.283} C_VEL
LIN {X 0,Y 247.738,Z 236.154,A -85,B 0,C 180,E1 -21198.665,E2 -21198.665} C_VEL
LIN {X 0,Y 241.57,Z 225.598,A -85,B 0,C 180,E1 -21200.875,E2 -21200.875} C_VEL
LIN {X 0,Y 234.513,Z 214.577,A -85,B 0,C 180,E1 -21203.643,E2 -21203.643} C_VEL
LIN {X 0,Y 227.663,Z 204.923,A -85,B 0,C 180,E1 -21206.641,E2 -21206.641} C_VEL
LIN {X 0,Y 223.532,Z 199.665,A -85,B 0,C 180,E1 -21208.636,E2 -21208.636} C_VEL
LIN {X 0,Y 217.028,Z 191.613,A -85,B 0,C 180,E1 -21212.198,E2 -21212.198} C_VEL
LIN {X 0,Y 213.664,Z 187.748,A -85,B 0,C 180,E1 -21214.293,E2 -21214.293} C_VEL
LIN {X 0,Y 212.489,Z 185.847,A -85,B 0,C 180,E1 -21215.58,E2 -21215.58} C_VEL
LIN {X 0,Y 210.882,Z 183.691,A -85,B 0,C 180,E1 -21217.464,E2 -21217.464} C_VEL
LIN {X 0,Y 210.34,Z 182.242,A -85,B 0,C 180,E1 -21218.436,E2 -21218.436} C_VEL
LIN {X 0,Y 207.145,Z 177.517,A -85,B 0,C 180,E1 -21223.238,E2 -21223.238} C_VEL
LIN {X 0,Y 206.869,Z 176.341,A -85,B 0,C 180,E1 -21224.229,E2 -21224.229} C_VEL
LIN {X 0,Y 207.124,Z 176.311,A -85,B 0,C 180,E1 -21230.232,E2 -21230.232} C_VEL
LIN {X 0,Y 207.065,Z 176.284,A -85,B 0,C 180,E1 -21234.156,E2 -21234.156} C_VEL
LIN {X 0,Y 207.374,Z 176.261,A -85,B 0,C 180,E1 -21238.058,E2 -21238.058} C_VEL
LIN {X 0,Y 207.418,Z 176.239,A -85,B 0,C 180,E1 -21240.888,E2 -21240.888} C_VEL
LIN {X 0,Y 206.68,Z 176.527,A -85,B 0,C 180,E1 -21242.504,E2 -21242.504} C_VEL
LIN {X 0,Y 203.952,Z 177.846,A -85,B 0,C 180,E1 -21245.136,E2 -21245.136} C_VEL
LIN {X 0,Y 201.933,Z 179.281,A -85,B 0,C 180,E1 -21247.276,E2 -21247.276} C_VEL
LIN {X 0,Y 201.415,Z 180.364,A -85,B 0,C 180,E1 -21248.927,E2 -21248.927} C_VEL
LIN {X 0,Y 201.554,Z 180.696,A -85,B 0,C 180,E1 -21249.479,E2 -21249.479} C_VEL
LIN {X 0,Y 204.08,Z 183.437,A -85,B 0,C 180,E1 -21253.949,E2 -21253.949} C_VEL
LIN {X 0,Y 205.178,Z 185.718,A -85,B 0,C 180,E1 -21255.904,E2 -21255.904} C_VEL
LIN {X 0,Y 207.538,Z 188.434,A -85,B 0,C 180,E1 -21258.766,E2 -21258.766} C_VEL
LIN {X 0,Y 209.063,Z 191.225,A -85,B 0,C 180,E1 -21260.669,E2 -21260.669} C_VEL
LIN {X 0,Y 211.014,Z 193.439,A -85,B 0,C 180,E1 -21262.521,E2 -21262.521} C_VEL
LIN {X 0,Y 214.021,Z 197.872,A -85,B 0,C 180,E1 -21265.27,E2 -21265.27} C_VEL
LIN {X 0,Y 217.559,Z 203.097,A -85,B 0,C 180,E1 -21267.981,E2 -21267.981} C_VEL
LIN {X 0,Y 223.395,Z 210.945,A -85,B 0,C 180,E1 -21271.109,E2 -21271.109} C_VEL
LIN {X 0,Y 229.069,Z 218.889,A -85,B 0,C 180,E1 -21273.785,E2 -21273.785} C_VEL
LIN {X 0,Y 234.343,Z 227.003,A -85,B 0,C 180,E1 -21276.048,E2 -21276.048} C_VEL
LIN {X 0,Y 239.685,Z 240.875,A -85,B 0,C 180,E1 -21278.394,E2 -21278.394} C_VEL
LIN {X 0,Y 245.859,Z 258.215,A -85,B 0,C 180,E1 -21280.903,E2 -21280.903} C_VEL
LIN {X 0,Y 247.494,Z 291.26,A -85,B 0,C 180,E1 -21282.72,E2 -21282.72} C_VEL
LIN {X 0,Y 241.94,Z 381.302,A -85,B 0,C 180,E1 -21285.147,E2 -21285.147} C_VEL
LIN {X 0,Y 239.957,Z 396.832,A -85,B 0,C 180,E1 -21285.782,E2 -21285.782} C_VEL
LIN {X 0,Y 237.354,Z 411.124,A -85,B 0,C 180,E1 -21286.644,E2 -21286.644} C_VEL
LIN {X 0,Y 234.023,Z 425.238,A -85,B 0,C 180,E1 -21287.786,E2 -21287.786} C_VEL
LIN {X 0,Y 230.076,Z 439.015,A -85,B 0,C 180,E1 -21289.241,E2 -21289.241} C_VEL
LIN {X 0,Y 225.891,Z 451.687,A -85,B 0,C 180,E1 -21290.953,E2 -21290.953} C_VEL
LIN {X 0,Y 221.206,Z 464.513,A -85,B 0,C 180,E1 -21293.156,E2 -21293.156} C_VEL
LIN {X 0,Y 216.778,Z 475.255,A -85,B 0,C 180,E1 -21295.437,E2 -21295.437} C_VEL
LIN {X 0,Y 212.591,Z 485.231,A -85,B 0,C 180,E1 -21298.069,E2 -21298.069} C_VEL
LIN {X 0,Y 208.871,Z 493.757,A -85,B 0,C 180,E1 -21300.802,E2 -21300.802} C_VEL
